LIN {X 0,Y 373.483,Z 447.363,A -85,B 0,C 180,E1 -12862.635,E2 -12862.635} C_VEL
LIN {X 0,Y 372.77,Z 459.424,A -85,B 0,C 180,E1 -12863.505,E2 -12863.505} C_VEL
LIN {X 0,Y 371.923,Z 468.35,A -85,B 0,C 180,E1 -12864.307,E2 -12864.307} C_VEL
LIN {X 0,Y 371.061,Z 479.116,A -85,B 0,C 180,E1 -12865.519,E2 -12865.519} C_VEL
LIN {X 0,Y 370.222,Z 487.926,A -85,B 0,C 180,E1 -12866.736,E2 -12866.736} C_VEL
LIN {X 0,Y 369.443,Z 497.479,A -85,B 0,C 180,E1 -12868.365,E2 -12868.365} C_VEL
LIN {X 0,Y 368.694,Z 505.108,A -85,B 0,C 180,E1 -12870,E2 -12870} C_VEL
LIN {X 0,Y 368.224,Z 511.231,A -85,B 0,C 180,E1 -12871.641,E2 -12871.641} C_VEL
LIN {X 0,Y 367.89,Z 516.098,A -85,B 0,C 180,E1 -12873.286,E2 -12873.286} C_VEL
LIN {X 0,Y 367.719,Z 519.853,A -85,B 0,C 180,E1 -12874.934,E2 -12874.934} C_VEL
LIN {X 0,Y 367.623,Z 522.596,A -85,B 0,C 180,E1 -12876.587,E2 -12876.587} C_VEL
LIN {X 0,Y 367.369,Z 524.811,A -85,B 0,C 180,E1 -12878.804,E2 -12878.804} C_VEL
LIN {X 0,Y 367.305,Z 525.292,A -85,B 0,C 180,E1 -12879.916,E2 -12879.916} C_VEL
LIN {X 0,Y 367.371,Z 525.357,A -85,B 0,C 180,E1 -12881.029,E2 -12881.029} C_VEL
LIN {X 0,Y 367.515,Z 524.674,A -85,B 0,C 180,E1 -12882.768,E2 -12882.768} C_VEL
LIN {X 0,Y 367.623,Z 523.153,A -85,B 0,C 180,E1 -12884.391,E2 -12884.391} C_VEL
LIN {X 0,Y 367.976,Z 520.609,A -85,B 0,C 180,E1 -12886.078,E2 -12886.078} C_VEL
LIN {X 0,Y 368.384,Z 517.012,A -85,B 0,C 180,E1 -12887.773,E2 -12887.773} C_VEL
LIN {X 0,Y 368.981,Z 512.245,A -85,B 0,C 180,E1 -12889.471,E2 -12889.471} C_VEL
LIN {X 0,Y 369.433,Z 508.887,A -85,B 0,C 180,E1 -12890.455,E2 -12890.455} C_VEL
LIN {X 0,Y 369.179,Z 505.977,A -85,B 0,C 180,E1 -12891.251,E2 -12891.251} C_VEL
LIN {X 0,Y 367.085,Z 500.999,A -85,B 0,C 180,E1 -12892.546,E2 -12892.546} C_VEL
LIN {X 0,Y 365.06,Z 495.431,A -85,B 0,C 180,E1 -12893.789,E2 -12893.789} C_VEL
LIN {X 0,Y 364.906,Z 491.596,A -85,B 0,C 180,E1 -12894.493,E2 -12894.493} C_VEL
LIN {X 0,Y 366.14,Z 482.192,A -85,B 0,C 180,E1 -12895.916,E2 -12895.916} C_VEL
LIN {X 0,Y 367.366,Z 471.755,A -85,B 0,C 180,E1 -12897.178,E2 -12897.178} C_VEL
LIN {X 0,Y 368.601,Z 459.913,A -85,B 0,C 180,E1 -12898.313,E2 -12898.313} C_VEL
LIN {X 0,Y 369.641,Z 447.439,A -85,B 0,C 180,E1 -12899.223,E2 -12899.223} C_VEL
LIN {X 0,Y 370.361,Z 434.476,A -85,B 0,C 180,E1 -12899.915,E2 -12899.915} C_VEL
LIN {X 0,Y 370.809,Z 422.498,A -85,B 0,C 180,E1 -12900.346,E2 -12900.346} C_VEL
LIN {X 0,Y 372.684,Z 341.338,A -85,B 0,C 180,E1 -12901.941,E2 -12901.941} C_VEL
LIN {X 0,Y 369.707,Z 328.526,A -85,B 0,C 180,E1 -12902.432,E2 -12902.432} C_VEL
LIN {X 0,Y 364.874,Z 317.06,A -85,B 0,C 180,E1 -12903.049,E2 -12903.049} C_VEL
LIN {X 0,Y 364.019,Z 314.785,A -85,B 0,C 180,E1 -12903.186,E2 -12903.186} C_VEL
LIN {X 0,Y 361.887,Z 305.411,A -85,B 0,C 180,E1 -12905.892,E2 -12905.892} C_VEL
LIN {X 0,Y 361.869,Z 305.412,A -85,B 0,C 180,E1 -12909.027,E2 -12909.027} C_VEL
LIN {X 0,Y 361.835,Z 305.415,A -85,B 0,C 180,E1 -12912.829,E2 -12912.829} C_VEL
LIN {X 0,Y 361.818,Z 305.415,A -85,B 0,C 180,E1 -12915.947,E2 -12915.947} C_VEL
LIN {X 0,Y 361.835,Z 305.412,A -85,B 0,C 180,E1 -12919.245,E2 -12919.245} C_VEL
LIN {X 0,Y 361.863,Z 305.409,A -85,B 0,C 180,E1 -12922.777,E2 -12922.777} C_VEL
LIN {X 0,Y 361.853,Z 305.404,A -85,B 0,C 180,E1 -12925.72,E2 -12925.72} C_VEL
LIN {X 0,Y 361.874,Z 305.401,A -85,B 0,C 180,E1 -12929.672,E2 -12929.672} C_VEL
LIN {X 0,Y 361.953,Z 305.392,A -85,B 0,C 180,E1 -12933.475,E2 -12933.475} C_VEL
LIN {X 0,Y 361.882,Z 305.399,A -85,B 0,C 180,E1 -12937.144,E2 -12937.144} C_VEL
LIN {X 0,Y 361.911,Z 305.393,A -85,B 0,C 180,E1 -12940.724,E2 -12940.724} C_VEL
LIN {X 0,Y 361.933,Z 305.4,A -85,B 0,C 180,E1 -12943.066,E2 -12943.066} C_VEL
LIN {X 0,Y 361.998,Z 305.39,A -85,B 0,C 180,E1 -12946.528,E2 -12946.528} C_VEL
LIN {X 0,Y 362.031,Z 305.387,A -85,B 0,C 180,E1 -12949.938,E2 -12949.938} C_VEL
LIN {X 0,Y 362.15,Z 305.37,A -85,B 0,C 180,E1 -12952.193,E2 -12952.193} C_VEL
LIN {X 0,Y 362.116,Z 305.375,A -85,B 0,C 180,E1 -12954.431,E2 -12954.431} C_VEL
LIN {X 0,Y 362.28,Z 305.352,A -85,B 0,C 180,E1 -12957.777,E2 -12957.777} C_VEL
LIN {X 0,Y 362.426,Z 305.34,A -85,B 0,C 180,E1 -12960,E2 -12960} C_VEL
LIN {X 0,Y 362.28,Z 305.35,A -85,B 0,C 180,E1 -12962.224,E2 -12962.224} C_VEL
LIN {X 0,Y 362.17,Z 305.361,A -85,B 0,C 180,E1 -12966.686,E2 -12966.686} C_VEL
LIN {X 0,Y 362.074,Z 305.38,A -85,B 0,C 180,E1 -12968.933,E2 -12968.933} C_VEL
LIN {X 0,Y 361.96,Z 305.39,A -85,B 0,C 180,E1 -12972.333,E2 -12972.333} C_VEL
LIN {X 0,Y 361.962,Z 305.394,A -85,B 0,C 180,E1 -12974.621,E2 -12974.621} C_VEL
LIN {X 0,Y 361.96,Z 305.395,A -85,B 0,C 180,E1 -12978.1,E2 -12978.1} C_VEL
LIN {X 0,Y 361.862,Z 305.405,A -85,B 0,C 180,E1 -12981.655,E2 -12981.655} C_VEL
LIN {X 0,Y 361.928,Z 305.399,A -85,B 0,C 180,E1 -12985.29,E2 -12985.29} C_VEL
LIN {X 0,Y 361.915,Z 305.398,A -85,B 0,C 180,E1 -12987.779,E2 -12987.779} C_VEL
LIN {X 0,Y 361.847,Z 305.409,A -85,B 0,C 180,E1 -12991.285,E2 -12991.285} C_VEL
LIN {X 0,Y 361.855,Z 305.408,A -85,B 0,C 180,E1 -12994.281,E2 -12994.281} C_VEL
LIN {X 0,Y 361.864,Z 305.41,A -85,B 0,C 180,E1 -12997.223,E2 -12997.223} C_VEL
LIN {X 0,Y 361.836,Z 305.393,A -85,B 0,C 180,E1 -13000.755,E2 -13000.755} C_VEL
LIN {X 0,Y 361.818,Z 305.41,A -85,B 0,C 180,E1 -13004.369,E2 -13004.369} C_VEL
LIN {X 0,Y 361.838,Z 305.415,A -85,B 0,C 180,E1 -13007.568,E2 -13007.568} C_VEL
LIN {X 0,Y 361.87,Z 305.407,A -85,B 0,C 180,E1 -13010.974,E2 -13010.974} C_VEL
LIN {X 0,Y 361.876,Z 305.408,A -85,B 0,C 180,E1 -13014.655,E2 -13014.655} C_VEL
LIN {X 0,Y 361.84,Z 305.414,A -85,B 0,C 180,E1 -13018.371,E2 -13018.371} C_VEL
LIN {X 0,Y 361.876,Z 305.581,A -85,B 0,C 180,E1 -13018.596,E2 -13018.596} C_VEL
LIN {X 0,Y 364.465,Z 316.266,A -85,B 0,C 180,E1 -13021.494,E2 -13021.494} C_VEL
LIN {X 0,Y 366.316,Z 325.27,A -85,B 0,C 180,E1 -13023.815,E2 -13023.815} C_VEL
LIN {X 0,Y 366.607,Z 328.794,A -85,B 0,C 180,E1 -13024.67,E2 -13024.67} C_VEL
LIN {X 0,Y 365.489,Z 339.127,A -85,B 0,C 180,E1 -13027.004,E2 -13027.004} C_VEL
LIN {X 0,Y 370.301,Z 363.459,A -85,B 0,C 180,E1 -13027.884,E2 -13027.884} C_VEL
LIN {X 0,Y 372.048,Z 374.943,A -85,B 0,C 180,E1 -13028.251,E2 -13028.251} C_VEL
LIN {X 0,Y 370.652,Z 448.342,A -85,B 0,C 180,E1 -13029.718,E2 -13029.718} C_VEL
LIN {X 0,Y 369.806,Z 462.108,A -85,B 0,C 180,E1 -13030.213,E2 -13030.213} C_VEL
LIN {X 0,Y 368.828,Z 474.473,A -85,B 0,C 180,E1 -13030.882,E2 -13030.882} C_VEL
LIN {X 0,Y 367.642,Z 486.322,A -85,B 0,C 180,E1 -13031.758,E2 -13031.758} C_VEL
LIN {X 0,Y 366.31,Z 497.713,A -85,B 0,C 180,E1 -13032.843,E2 -13032.843} C_VEL
LIN {X 0,Y 365.033,Z 508.003,A -85,B 0,C 180,E1 -13034.076,E2 -13034.076} C_VEL
LIN {X 0,Y 363.946,Z 517.267,A -85,B 0,C 180,E1 -13035.461,E2 -13035.461} C_VEL
LIN {X 0,Y 362.775,Z 526.272,A -85,B 0,C 180,E1 -13037.127,E2 -13037.127} C_VEL
LIN {X 0,Y 361.748,Z 533.548,A -85,B 0,C 180,E1 -13038.797,E2 -13038.797} C_VEL
LIN {X 0,Y 361.097,Z 539.398,A -85,B 0,C 180,E1 -13040.477,E2 -13040.477} C_VEL
LIN {X 0,Y 360.68,Z 544.022,A -85,B 0,C 180,E1 -13042.16,E2 -13042.16} C_VEL
LIN {X 0,Y 360.433,Z 547.766,A -85,B 0,C 180,E1 -13043.956,E2 -13043.956} C_VEL
LIN {X 0,Y 360.366,Z 550.098,A -85,B 0,C 180,E1 -13045.525,E2 -13045.525} C_VEL
LIN {X 0,Y 360.302,Z 551.291,A -85,B 0,C 180,E1 -13046.645,E2 -13046.645} C_VEL
LIN {X 0,Y 360.359,Z 552.416,A -85,B 0,C 180,E1 -13048.882,E2 -13048.882} C_VEL
LIN {X 0,Y 360.423,Z 552.399,A -85,B 0,C 180,E1 -13050,E2 -13050} C_VEL
LIN {X 0,Y 360.39,Z 551.989,A -85,B 0,C 180,E1 -13051.117,E2 -13051.117} C_VEL
LIN {X 0,Y 360.326,Z 551.137,A -85,B 0,C 180,E1 -13052.235,E2 -13052.235} C_VEL
LIN {X 0,Y 360.323,Z 549.88,A -85,B 0,C 180,E1 -13053.354,E2 -13053.354} C_VEL
LIN {X 0,Y 360.38,Z 547.205,A -85,B 0,C 180,E1 -13055.034,E2 -13055.034} C_VEL
LIN {X 0,Y 360.498,Z 543.495,A -85,B 0,C 180,E1 -13056.717,E2 -13056.717} C_VEL
LIN {X 0,Y 360.74,Z 538.65,A -85,B 0,C 180,E1 -13058.401,E2 -13058.401} C_VEL
LIN {X 0,Y 361.156,Z 532.524,A -85,B 0,C 180,E1 -13060.086,E2 -13060.086} C_VEL
LIN {X 0,Y 361.781,Z 524.896,A -85,B 0,C 180,E1 -13061.769,E2 -13061.769} C_VEL
LIN {X 0,Y 362.498,Z 517.094,A -85,B 0,C 180,E1 -13063.167,E2 -13063.167} C_VEL
LIN {X 0,Y 363.408,Z 507.556,A -85,B 0,C 180,E1 -13064.56,E2 -13064.56} C_VEL
LIN {X 0,Y 364.157,Z 496.934,A -85,B 0,C 180,E1 -13065.819,E2 -13065.819} C_VEL
LIN {X 0,Y 365.223,Z 485.127,A -85,B 0,C 180,E1 -13066.92,E2 -13066.92} C_VEL
LIN {X 0,Y 366.096,Z 473.602,A -85,B 0,C 180,E1 -13067.743,E2 -13067.743} C_VEL
LIN {X 0,Y 366.89,Z 460.601,A -85,B 0,C 180,E1 -13068.425,E2 -13068.425} C_VEL
LIN {X 0,Y 367.493,Z 448.03,A -85,B 0,C 180,E1 -13068.863,E2 -13068.863} C_VEL
LIN {X 0,Y 368.551,Z 374.347,A -85,B 0,C 180,E1 -13070.314,E2 -13070.314} C_VEL
LIN {X 0,Y 363.817,Z 339.576,A -85,B 0,C 180,E1 -13071.265,E2 -13071.265} C_VEL
LIN {X 0,Y 365.161,Z 323.765,A -85,B 0,C 180,E1 -13074.746,E2 -13074.746} C_VEL
LIN {X 0,Y 364.791,Z 319.684,A -85,B 0,C 180,E1 -13075.692,E2 -13075.692} C_VEL
LIN {X 0,Y 362.335,Z 307.335,A -85,B 0,C 180,E1 -13078.689,E2 -13078.689} C_VEL
LIN {X 0,Y 361.935,Z 305.401,A -85,B 0,C 180,E1 -13079.184,E2 -13079.184} C_VEL
LIN {X 0,Y 361.858,Z 305.406,A -85,B 0,C 180,E1 -13083.369,E2 -13083.369} C_VEL
LIN {X 0,Y 361.866,Z 305.406,A -85,B 0,C 180,E1 -13087.017,E2 -13087.017} C_VEL
LIN {X 0,Y 361.853,Z 305.409,A -85,B 0,C 180,E1 -13089.861,E2 -13089.861} C_VEL
LIN {X 0,Y 361.834,Z 305.412,A -85,B 0,C 180,E1 -13092.828,E2 -13092.828} C_VEL
LIN {X 0,Y 361.816,Z 305.413,A -85,B 0,C 180,E1 -13095.946,E2 -13095.946} C_VEL
LIN {X 0,Y 361.833,Z 305.41,A -85,B 0,C 180,E1 -13099.244,E2 -13099.244} C_VEL
LIN {X 0,Y 361.861,Z 305.412,A -85,B 0,C 180,E1 -13102.776,E2 -13102.776} C_VEL
LIN {X 0,Y 361.851,Z 305.407,A -85,B 0,C 180,E1 -13105.719,E2 -13105.719} C_VEL
LIN {X 0,Y 361.869,Z 305.405,A -85,B 0,C 180,E1 -13109.671,E2 -13109.671} C_VEL
LIN {X 0,Y 361.95,Z 305.397,A -85,B 0,C 180,E1 -13113.474,E2 -13113.474} C_VEL
LIN {X 0,Y 361.886,Z 305.409,A -85,B 0,C 180,E1 -13117.144,E2 -13117.144} C_VEL
LIN {X 0,Y 361.917,Z 305.401,A -85,B 0,C 180,E1 -13120.724,E2 -13120.724} C_VEL
LIN {X 0,Y 361.942,Z 305.396,A -85,B 0,C 180,E1 -13124.226,E2 -13124.226} C_VEL
LIN {X 0,Y 361.994,Z 305.389,A -85,B 0,C 180,E1 -13126.527,E2 -13126.527} C_VEL
LIN {X 0,Y 362.027,Z 305.387,A -85,B 0,C 180,E1 -13129.938,E2 -13129.938} C_VEL
LIN {X 0,Y 362.157,Z 305.373,A -85,B 0,C 180,E1 -13133.313,E2 -13133.313} C_VEL
LIN {X 0,Y 362.275,Z 305.36,A -85,B 0,C 180,E1 -13137.776,E2 -13137.776} C_VEL
LIN {X 0,Y 362.421,Z 305.34,A -85,B 0,C 180,E1 -13140,E2 -13140} C_VEL
LIN {X 0,Y 362.276,Z 305.356,A -85,B 0,C 180,E1 -13142.223,E2 -13142.223} C_VEL
LIN {X 0,Y 362.134,Z 305.372,A -85,B 0,C 180,E1 -13146.687,E2 -13146.687} C_VEL
LIN {X 0,Y 362.026,Z 305.392,A -85,B 0,C 180,E1 -13150.062,E2 -13150.062} C_VEL
LIN {X 0,Y 361.993,Z 305.394,A -85,B 0,C 180,E1 -13153.899,E2 -13153.899} C_VEL
LIN {X 0,Y 361.962,Z 305.397,A -85,B 0,C 180,E1 -13157.939,E2 -13157.939} C_VEL
LIN {X 0,Y 361.856,Z 305.407,A -85,B 0,C 180,E1 -13161.655,E2 -13161.655} C_VEL
LIN {X 0,Y 361.921,Z 305.399,A -85,B 0,C 180,E1 -13165.29,E2 -13165.29} C_VEL
LIN {X 0,Y 361.913,Z 305.4,A -85,B 0,C 180,E1 -13167.778,E2 -13167.778} C_VEL
LIN {X 0,Y 361.842,Z 305.409,A -85,B 0,C 180,E1 -13171.285,E2 -13171.285} C_VEL
LIN {X 0,Y 361.849,Z 305.41,A -85,B 0,C 180,E1 -13174.281,E2 -13174.281} C_VEL
LIN {X 0,Y 361.858,Z 305.408,A -85,B 0,C 180,E1 -13177.223,E2 -13177.223} C_VEL
LIN {X 0,Y 361.831,Z 305.416,A -85,B 0,C 180,E1 -13180.756,E2 -13180.756} C_VEL
LIN {X 0,Y 361.812,Z 305.413,A -85,B 0,C 180,E1 -13184.369,E2 -13184.369} C_VEL
LIN {X 0,Y 361.825,Z 305.412,A -85,B 0,C 180,E1 -13187.57,E2 -13187.57} C_VEL
LIN {X 0,Y 361.84,Z 305.411,A -85,B 0,C 180,E1 -13191.573,E2 -13191.573} C_VEL
LIN {X 0,Y 361.871,Z 305.406,A -85,B 0,C 180,E1 -13194.656,E2 -13194.656} C_VEL
LIN {X 0,Y 361.834,Z 305.409,A -85,B 0,C 180,E1 -13198.371,E2 -13198.371} C_VEL
LIN {X 0,Y 361.863,Z 305.408,A -85,B 0,C 180,E1 -13200.953,E2 -13200.953} C_VEL
LIN {X 0,Y 361.863,Z 305.406,A -85,B 0,C 180,E1 -13204.706,E2 -13204.706} C_VEL
LIN {X 0,Y 361.859,Z 305.407,A -85,B 0,C 180,E1 -13208.346,E2 -13208.346} C_VEL
LIN {X 0,Y 361.919,Z 305.401,A -85,B 0,C 180,E1 -13212.085,E2 -13212.085} C_VEL
LIN {X 0,Y 361.961,Z 305.397,A -85,B 0,C 180,E1 -13215.38,E2 -13215.38} C_VEL
LIN {X 0,Y 362.044,Z 305.52,A -85,B 0,C 180,E1 -13216.471,E2 -13216.471} C_VEL
LIN {X 0,Y 363.735,Z 314.698,A -85,B 0,C 180,E1 -13218.825,E2 -13218.825} C_VEL
LIN {X 0,Y 366.129,Z 323.28,A -85,B 0,C 180,E1 -13219.123,E2 -13219.123} C_VEL
LIN {X 0,Y 369.003,Z 340.775,A -85,B 0,C 180,E1 -13219.62,E2 -13219.62} C_VEL
LIN {X 0,Y 367.65,Z 421.709,A -85,B 0,C 180,E1 -13221.204,E2 -13221.204} C_VEL
LIN {X 0,Y 367.211,Z 434.918,A -85,B 0,C 180,E1 -13221.678,E2 -13221.678} C_VEL
LIN {X 0,Y 366.63,Z 447.574,A -85,B 0,C 180,E1 -13222.358,E2 -13222.358} C_VEL
LIN {X 0,Y 365.897,Z 459.648,A -85,B 0,C 180,E1 -13223.244,E2 -13223.244} C_VEL
LIN {X 0,Y 365.012,Z 468.583,A -85,B 0,C 180,E1 -13224.06,E2 -13224.06} C_VEL
LIN {X 0,Y 364.125,Z 479.354,A -85,B 0,C 180,E1 -13225.295,E2 -13225.295} C_VEL
LIN {X 0,Y 363.193,Z 489.05,A -85,B 0,C 180,E1 -13226.672,E2 -13226.672} C_VEL
LIN {X 0,Y 362.499,Z 496.99,A -85,B 0,C 180,E1 -13228.056,E2 -13228.056} C_VEL
LIN {X 0,Y 361.721,Z 504.802,A -85,B 0,C 180,E1 -13229.722,E2 -13229.722} C_VEL
LIN {X 0,Y 361.258,Z 510.097,A -85,B 0,C 180,E1 -13231.115,E2 -13231.115} C_VEL
LIN {X 0,Y 360.914,Z 515.27,A -85,B 0,C 180,E1 -13232.791,E2 -13232.791} C_VEL
LIN {X 0,Y 360.627,Z 519.299,A -85,B 0,C 180,E1 -13234.471,E2 -13234.471} C_VEL
LIN {X 0,Y 360.589,Z 522.465,A -85,B 0,C 180,E1 -13236.278,E2 -13236.278} C_VEL
LIN {X 0,Y 360.357,Z 524.306,A -85,B 0,C 180,E1 -13237.847,E2 -13237.847} C_VEL
LIN {X 0,Y 360.255,Z 525.162,A -85,B 0,C 180,E1 -13238.979,E2 -13238.979} C_VEL
LIN {X 0,Y 360.314,Z 525.604,A -85,B 0,C 180,E1 -13241.248,E2 -13241.248} C_VEL
LIN {X 0,Y 360.443,Z 524.953,A -85,B 0,C 180,E1 -13242.862,E2 -13242.862} C_VEL
LIN {X 0,Y 360.598,Z 523.239,A -85,B 0,C 180,E1 -13244.677,E2 -13244.677} C_VEL
LIN {X 0,Y 360.959,Z 520.611,A -85,B 0,C 180,E1 -13246.399,E2 -13246.399} C_VEL
LIN {X 0,Y 361.435,Z 516.923,A -85,B 0,C 180,E1 -13248.127,E2 -13248.127} C_VEL
LIN {X 0,Y 362.065,Z 512.058,A -85,B 0,C 180,E1 -13249.858,E2 -13249.858} C_VEL
LIN {X 0,Y 362.941,Z 505.631,A -85,B 0,C 180,E1 -13251.648,E2 -13251.648} C_VEL
LIN {X 0,Y 363.969,Z 498.087,A -85,B 0,C 180,E1 -13253.319,E2 -13253.319} C_VEL
LIN {X 0,Y 364.906,Z 491.596,A -85,B 0,C 180,E1 -13254.493,E2 -13254.493} C_VEL
LIN {X 0,Y 364.796,Z 487.582,A -85,B 0,C 180,E1 -13255.176,E2 -13255.176} C_VEL
LIN {X 0,Y 362.993,Z 480.92,A -85,B 0,C 180,E1 -13256.299,E2 -13256.299} C_VEL
LIN {X 0,Y 361.199,Z 473.773,A -85,B 0,C 180,E1 -13257.344,E2 -13257.344} C_VEL
LIN {X 0,Y 361.086,Z 469.006,A -85,B 0,C 180,E1 -13257.894,E2 -13257.894} C_VEL
LIN {X 0,Y 362.176,Z 458.535,A -85,B 0,C 180,E1 -13258.862,E2 -13258.862} C_VEL
LIN {X 0,Y 363.184,Z 446.482,A -85,B 0,C 180,E1 -13259.726,E2 -13259.726} C_VEL
LIN {X 0,Y 363.944,Z 433.308,A -85,B 0,C 180,E1 -13260.418,E2 -13260.418} C_VEL
LIN {X 0,Y 364.313,Z 422.973,A -85,B 0,C 180,E1 -13260.785,E2 -13260.785} C_VEL
LIN {X 0,Y 366.246,Z 342.244,A -85,B 0,C 180,E1 -13262.4,E2 -13262.4} C_VEL
LIN {X 0,Y 363.71,Z 331.264,A -85,B 0,C 180,E1 -13262.832,E2 -13262.832} C_VEL
LIN {X 0,Y 356.879,Z 315.033,A -85,B 0,C 180,E1 -13263.772,E2 -13263.772} C_VEL
LIN {X 0,Y 354.848,Z 306.282,A -85,B 0,C 180,E1 -13266.35,E2 -13266.35} C_VEL
LIN {X 0,Y 354.824,Z 306.288,A -85,B 0,C 180,E1 -13269.424,E2 -13269.424} C_VEL
LIN {X 0,Y 354.787,Z 306.293,A -85,B 0,C 180,E1 -13272.867,E2 -13272.867} C_VEL
LIN {X 0,Y 354.766,Z 306.294,A -85,B 0,C 180,E1 -13276.104,E2 -13276.104} C_VEL
LIN {X 0,Y 354.788,Z 306.29,A -85,B 0,C 180,E1 -13279.179,E2 -13279.179} C_VEL
LIN {X 0,Y 354.807,Z 306.285,A -85,B 0,C 180,E1 -13282.403,E2 -13282.403} C_VEL
LIN {X 0,Y 354.811,Z 306.285,A -85,B 0,C 180,E1 -13284.941,E2 -13284.941} C_VEL
LIN {X 0,Y 354.793,Z 306.283,A -85,B 0,C 180,E1 -13288.405,E2 -13288.405} C_VEL
LIN {X 0,Y 354.848,Z 306.274,A -85,B 0,C 180,E1 -13291.619,E2 -13291.619} C_VEL
LIN {X 0,Y 354.898,Z 306.27,A -85,B 0,C 180,E1 -13294.173,E2 -13294.173} C_VEL
LIN {X 0,Y 354.816,Z 306.284,A -85,B 0,C 180,E1 -13297.893,E2 -13297.893} C_VEL
LIN {X 0,Y 354.922,Z 306.274,A -85,B 0,C 180,E1 -13301.892,E2 -13301.892} C_VEL
LIN {X 0,Y 354.943,Z 306.272,A -85,B 0,C 180,E1 -13305.981,E2 -13305.981} C_VEL
LIN {X 0,Y 354.977,Z 306.263,A -85,B 0,C 180,E1 -13309.736,E2 -13309.736} C_VEL
LIN {X 0,Y 355.113,Z 306.248,A -85,B 0,C 180,E1 -13312.037,E2 -13312.037} C_VEL
LIN {X 0,Y 355.091,Z 306.251,A -85,B 0,C 180,E1 -13314.321,E2 -13314.321} C_VEL
LIN {X 0,Y 355.244,Z 306.228,A -85,B 0,C 180,E1 -13317.733,E2 -13317.733} C_VEL
LIN {X 0,Y 355.375,Z 306.218,A -85,B 0,C 180,E1 -13320,E2 -13320} C_VEL
LIN {X 0,Y 355.243,Z 306.226,A -85,B 0,C 180,E1 -13322.268,E2 -13322.268} C_VEL
LIN {X 0,Y 355.137,Z 306.236,A -85,B 0,C 180,E1 -13326.819,E2 -13326.819} C_VEL
LIN {X 0,Y 355.015,Z 306.258,A -85,B 0,C 180,E1 -13329.113,E2 -13329.113} C_VEL
LIN {X 0,Y 354.921,Z 306.269,A -85,B 0,C 180,E1 -13332.581,E2 -13332.581} C_VEL
LIN {X 0,Y 354.89,Z 306.27,A -85,B 0,C 180,E1 -13336.096,E2 -13336.096} C_VEL
LIN {X 0,Y 354.907,Z 306.277,A -85,B 0,C 180,E1 -13338.472,E2 -13338.472} C_VEL
LIN {X 0,Y 354.818,Z 306.284,A -85,B 0,C 180,E1 -13342.107,E2 -13342.107} C_VEL
LIN {X 0,Y 354.899,Z 306.273,A -85,B 0,C 180,E1 -13345.828,E2 -13345.828} C_VEL
LIN {X 0,Y 354.855,Z 306.28,A -85,B 0,C 180,E1 -13349.679,E2 -13349.679} C_VEL
LIN {X 0,Y 354.807,Z 306.287,A -85,B 0,C 180,E1 -13353.702,E2 -13353.702} C_VEL
LIN {X 0,Y 354.798,Z 306.283,A -85,B 0,C 180,E1 -13356.46,E2 -13356.46} C_VEL
LIN {X 0,Y 354.825,Z 306.271,A -85,B 0,C 180,E1 -13359.424,E2 -13359.424} C_VEL
LIN {X 0,Y 354.79,Z 306.289,A -85,B 0,C 180,E1 -13362.867,E2 -13362.867} C_VEL
LIN {X 0,Y 354.768,Z 306.292,A -85,B 0,C 180,E1 -13366.104,E2 -13366.104} C_VEL
LIN {X 0,Y 354.789,Z 306.29,A -85,B 0,C 180,E1 -13369.179,E2 -13369.179} C_VEL
LIN {X 0,Y 354.809,Z 306.282,A -85,B 0,C 180,E1 -13372.403,E2 -13372.403} C_VEL
LIN {X 0,Y 354.814,Z 306.286,A -85,B 0,C 180,E1 -13374.941,E2 -13374.941} C_VEL
LIN {X 0,Y 354.794,Z 306.387,A -85,B 0,C 180,E1 -13378.087,E2 -13378.087} C_VEL
LIN {X 0,Y 357.582,Z 317.605,A -85,B 0,C 180,E1 -13381.215,E2 -13381.215} C_VEL
LIN {X 0,Y 359.685,Z 328.237,A -85,B 0,C 180,E1 -13384.003,E2 -13384.003} C_VEL
LIN {X 0,Y 359.409,Z 333.05,A -85,B 0,C 180,E1 -13385.139,E2 -13385.139} C_VEL
LIN {X 0,Y 358.771,Z 338.826,A -85,B 0,C 180,E1 -13386.469,E2 -13386.469} C_VEL
LIN {X 0,Y 363.58,Z 362.705,A -85,B 0,C 180,E1 -13387.371,E2 -13387.371} C_VEL
LIN {X 0,Y 365.621,Z 376.5,A -85,B 0,C 180,E1 -13387.819,E2 -13387.819} C_VEL
LIN {X 0,Y 364.145,Z 447.901,A -85,B 0,C 180,E1 -13389.265,E2 -13389.265} C_VEL
LIN {X 0,Y 363.291,Z 461.72,A -85,B 0,C 180,E1 -13389.769,E2 -13389.769} C_VEL
LIN {X 0,Y 362.275,Z 474.114,A -85,B 0,C 180,E1 -13390.449,E2 -13390.449} C_VEL
LIN {X 0,Y 361.141,Z 485.193,A -85,B 0,C 180,E1 -13391.27,E2 -13391.27} C_VEL
LIN {X 0,Y 359.721,Z 496.737,A -85,B 0,C 180,E1 -13392.372,E2 -13392.372} C_VEL
LIN {X 0,Y 358.346,Z 507.144,A -85,B 0,C 180,E1 -13393.624,E2 -13393.624} C_VEL
LIN {X 0,Y 357.23,Z 515.967,A -85,B 0,C 180,E1 -13394.939,E2 -13394.939} C_VEL
LIN {X 0,Y 356.011,Z 524.944,A -85,B 0,C 180,E1 -13396.587,E2 -13396.587} C_VEL
LIN {X 0,Y 354.909,Z 532.405,A -85,B 0,C 180,E1 -13398.289,E2 -13398.289} C_VEL
LIN {X 0,Y 354.061,Z 539.321,A -85,B 0,C 180,E1 -13400.286,E2 -13400.286} C_VEL
LIN {X 0,Y 353.624,Z 543.903,A -85,B 0,C 180,E1 -13402.003,E2 -13402.003} C_VEL
LIN {X 0,Y 353.325,Z 547.893,A -85,B 0,C 180,E1 -13404.019,E2 -13404.019} C_VEL
LIN {X 0,Y 353.279,Z 549.911,A -85,B 0,C 180,E1 -13405.436,E2 -13405.436} C_VEL
LIN {X 0,Y 353.223,Z 551.073,A -85,B 0,C 180,E1 -13406.578,E2 -13406.578} C_VEL
LIN {X 0,Y 353.26,Z 552.159,A -85,B 0,C 180,E1 -13408.86,E2 -13408.86} C_VEL
LIN {X 0,Y 353.328,Z 552.126,A -85,B 0,C 180,E1 -13410,E2 -13410} C_VEL
LIN {X 0,Y 353.292,Z 551.688,A -85,B 0,C 180,E1 -13411.139,E2 -13411.139} C_VEL
LIN {X 0,Y 353.245,Z 549.537,A -85,B 0,C 180,E1 -13413.421,E2 -13413.421} C_VEL
LIN {X 0,Y 353.283,Z 546.823,A -85,B 0,C 180,E1 -13415.136,E2 -13415.136} C_VEL
LIN {X 0,Y 353.416,Z 543.073,A -85,B 0,C 180,E1 -13416.852,E2 -13416.852} C_VEL
LIN {X 0,Y 353.679,Z 538.186,A -85,B 0,C 180,E1 -13418.57,E2 -13418.57} C_VEL
LIN {X 0,Y 354.121,Z 532.014,A -85,B 0,C 180,E1 -13420.289,E2 -13420.289} C_VEL
LIN {X 0,Y 354.802,Z 524.33,A -85,B 0,C 180,E1 -13422.004,E2 -13422.004} C_VEL
LIN {X 0,Y 355.518,Z 516.45,A -85,B 0,C 180,E1 -13423.431,E2 -13423.431} C_VEL
LIN {X 0,Y 356.439,Z 506.815,A -85,B 0,C 180,E1 -13424.852,E2 -13424.852} C_VEL
LIN {X 0,Y 357.342,Z 496.108,A -85,B 0,C 180,E1 -13426.129,E2 -13426.129} C_VEL
LIN {X 0,Y 358.248,Z 485.776,A -85,B 0,C 180,E1 -13427.113,E2 -13427.113} C_VEL
LIN {X 0,Y 359.218,Z 473.482,A -85,B 0,C 180,E1 -13428.021,E2 -13428.021} C_VEL
LIN {X 0,Y 360.054,Z 460.535,A -85,B 0,C 180,E1 -13428.714,E2 -13428.714} C_VEL
LIN {X 0,Y 360.663,Z 448.059,A -85,B 0,C 180,E1 -13429.16,E2 -13429.16} C_VEL
LIN {X 0,Y 361.71,Z 373.95,A -85,B 0,C 180,E1 -13430.653,E2 -13430.653} C_VEL
LIN {X 0,Y 356.886,Z 339.268,A -85,B 0,C 180,E1 -13431.638,E2 -13431.638} C_VEL
LIN {X 0,Y 358.206,Z 324.519,A -85,B 0,C 180,E1 -13434.949,E2 -13434.949} C_VEL
LIN {X 0,Y 357.487,Z 319.076,A -85,B 0,C 180,E1 -13436.252,E2 -13436.252} C_VEL
LIN {X 0,Y 354.917,Z 306.486,A -85,B 0,C 180,E1 -13439.392,E2 -13439.392} C_VEL
LIN {X 0,Y 354.87,Z 306.281,A -85,B 0,C 180,E1 -13439.676,E2 -13439.676} C_VEL
LIN {X 0,Y 354.806,Z 306.287,A -85,B 0,C 180,E1 -13443.701,E2 -13443.701} C_VEL
LIN {X 0,Y 354.797,Z 306.29,A -85,B 0,C 180,E1 -13446.459,E2 -13446.459} C_VEL
LIN {X 0,Y 354.823,Z 306.283,A -85,B 0,C 180,E1 -13449.423,E2 -13449.423} C_VEL
LIN {X 0,Y 354.786,Z 306.29,A -85,B 0,C 180,E1 -13452.866,E2 -13452.866} C_VEL
LIN {X 0,Y 354.765,Z 306.292,A -85,B 0,C 180,E1 -13456.103,E2 -13456.103} C_VEL
LIN {X 0,Y 354.786,Z 306.289,A -85,B 0,C 180,E1 -13459.178,E2 -13459.178} C_VEL
LIN {X 0,Y 354.805,Z 306.288,A -85,B 0,C 180,E1 -13462.402,E2 -13462.402} C_VEL
LIN {X 0,Y 354.809,Z 306.289,A -85,B 0,C 180,E1 -13464.94,E2 -13464.94} C_VEL
LIN {X 0,Y 354.79,Z 306.289,A -85,B 0,C 180,E1 -13468.404,E2 -13468.404} C_VEL
LIN {X 0,Y 354.843,Z 306.281,A -85,B 0,C 180,E1 -13471.618,E2 -13471.618} C_VEL
LIN {X 0,Y 354.895,Z 306.274,A -85,B 0,C 180,E1 -13474.172,E2 -13474.172} C_VEL
LIN {X 0,Y 354.831,Z 306.282,A -85,B 0,C 180,E1 -13477.893,E2 -13477.893} C_VEL
LIN {X 0,Y 354.919,Z 306.271,A -85,B 0,C 180,E1 -13481.891,E2 -13481.891} C_VEL
LIN {X 0,Y 354.938,Z 306.269,A -85,B 0,C 180,E1 -13485.981,E2 -13485.981} C_VEL
LIN {X 0,Y 354.973,Z 306.267,A -85,B 0,C 180,E1 -13489.736,E2 -13489.736} C_VEL
LIN {X 0,Y 355.122,Z 306.248,A -85,B 0,C 180,E1 -13493.18,E2 -13493.18} C_VEL
LIN {X 0,Y 355.238,Z 306.237,A -85,B 0,C 180,E1 -13497.732,E2 -13497.732} C_VEL
LIN {X 0,Y 355.37,Z 306.218,A -85,B 0,C 180,E1 -13500,E2 -13500} C_VEL
LIN {X 0,Y 355.239,Z 306.233,A -85,B 0,C 180,E1 -13502.267,E2 -13502.267} C_VEL
LIN {X 0,Y 355.098,Z 306.248,A -85,B 0,C 180,E1 -13506.82,E2 -13506.82} C_VEL
LIN {X 0,Y 354.973,Z 306.268,A -85,B 0,C 180,E1 -13510.264,E2 -13510.264} C_VEL
LIN {X 0,Y 354.938,Z 306.274,A -85,B 0,C 180,E1 -13514.019,E2 -13514.019} C_VEL
LIN {X 0,Y 354.917,Z 306.276,A -85,B 0,C 180,E1 -13518.109,E2 -13518.109} C_VEL
LIN {X 0,Y 354.81,Z 306.289,A -85,B 0,C 180,E1 -13522.107,E2 -13522.107} C_VEL
LIN {X 0,Y 354.893,Z 306.275,A -85,B 0,C 180,E1 -13525.828,E2 -13525.828} C_VEL
LIN {X 0,Y 354.849,Z 306.28,A -85,B 0,C 180,E1 -13529.679,E2 -13529.679} C_VEL
LIN {X 0,Y 354.801,Z 306.285,A -85,B 0,C 180,E1 -13533.702,E2 -13533.702} C_VEL
LIN {X 0,Y 354.793,Z 306.29,A -85,B 0,C 180,E1 -13536.46,E2 -13536.46} C_VEL
LIN {X 0,Y 354.82,Z 306.284,A -85,B 0,C 180,E1 -13539.424,E2 -13539.424} C_VEL
LIN {X 0,Y 354.783,Z 306.294,A -85,B 0,C 180,E1 -13542.868,E2 -13542.868} C_VEL
LIN {X 0,Y 354.761,Z 306.29,A -85,B 0,C 180,E1 -13546.104,E2 -13546.104} C_VEL
LIN {X 0,Y 354.762,Z 306.296,A -85,B 0,C 180,E1 -13549.176,E2 -13549.176} C_VEL
LIN {X 0,Y 354.797,Z 306.286,A -85,B 0,C 180,E1 -13552.404,E2 -13552.404} C_VEL
LIN {X 0,Y 354.809,Z 306.288,A -85,B 0,C 180,E1 -13554.941,E2 -13554.941} C_VEL
LIN {X 0,Y 354.79,Z 306.287,A -85,B 0,C 180,E1 -13558.406,E2 -13558.406} C_VEL
LIN {X 0,Y 354.794,Z 306.291,A -85,B 0,C 180,E1 -13561.615,E2 -13561.615} C_VEL
LIN {X 0,Y 354.803,Z 306.291,A -85,B 0,C 180,E1 -13565.42,E2 -13565.42} C_VEL
LIN {X 0,Y 354.825,Z 306.284,A -85,B 0,C 180,E1 -13569.114,E2 -13569.114} C_VEL
LIN {X 0,Y 354.878,Z 306.276,A -85,B 0,C 180,E1 -13572.72,E2 -13572.72} C_VEL
LIN {X 0,Y 354.974,Z 306.412,A -85,B 0,C 180,E1 -13576.216,E2 -13576.216} C_VEL
LIN {X 0,Y 356.56,Z 314.765,A -85,B 0,C 180,E1 -13578.438,E2 -13578.438} C_VEL
LIN {X 0,Y 359.384,Z 324.267,A -85,B 0,C 180,E1 -13578.794,E2 -13578.794} C_VEL
LIN {X 0,Y 362.203,Z 340.303,A -85,B 0,C 180,E1 -13579.27,E2 -13579.27} C_VEL
LIN {X 0,Y 360.834,Z 422.967,A -85,B 0,C 180,E1 -13580.93,E2 -13580.93} C_VEL
LIN {X 0,Y 360.327,Z 436.611,A -85,B 0,C 180,E1 -13581.448,E2 -13581.448} C_VEL
LIN {X 0,Y 359.762,Z 448.868,A -85,B 0,C 180,E1 -13582.141,E2 -13582.141} C_VEL
LIN {X 0,Y 358.92,Z 461.44,A -85,B 0,C 180,E1 -13583.112,E2 -13583.112} C_VEL
LIN {X 0,Y 357.736,Z 472.684,A -85,B 0,C 180,E1 -13584.222,E2 -13584.222} C_VEL
LIN {X 0,Y 356.847,Z 482.758,A -85,B 0,C 180,E1 -13585.482,E2 -13585.482} C_VEL
LIN {X 0,Y 356.01,Z 491.835,A -85,B 0,C 180,E1 -13586.888,E2 -13586.888} C_VEL
LIN {X 0,Y 355.193,Z 500.684,A -85,B 0,C 180,E1 -13588.583,E2 -13588.583} C_VEL
LIN {X 0,Y 354.465,Z 507.825,A -85,B 0,C 180,E1 -13590.284,E2 -13590.284} C_VEL
LIN {X 0,Y 354.066,Z 512.637,A -85,B 0,C 180,E1 -13591.707,E2 -13591.707} C_VEL
LIN {X 0,Y 353.659,Z 517.326,A -85,B 0,C 180,E1 -13593.418,E2 -13593.418} C_VEL
LIN {X 0,Y 353.552,Z 520.902,A -85,B 0,C 180,E1 -13595.132,E2 -13595.132} C_VEL
LIN {X 0,Y 353.385,Z 523.486,A -85,B 0,C 180,E1 -13596.854,E2 -13596.854} C_VEL
LIN {X 0,Y 353.257,Z 524.709,A -85,B 0,C 180,E1 -13598.006,E2 -13598.006} C_VEL
LIN {X 0,Y 353.152,Z 525.489,A -85,B 0,C 180,E1 -13599.161,E2 -13599.161} C_VEL
LIN {X 0,Y 353.228,Z 525.851,A -85,B 0,C 180,E1 -13601.477,E2 -13601.477} C_VEL
LIN {X 0,Y 353.367,Z 525.236,A -85,B 0,C 180,E1 -13602.956,E2 -13602.956} C_VEL
LIN {X 0,Y 353.556,Z 523.327,A -85,B 0,C 180,E1 -13604.976,E2 -13604.976} C_VEL
LIN {X 0,Y 353.965,Z 520.613,A -85,B 0,C 180,E1 -13606.732,E2 -13606.732} C_VEL
LIN {X 0,Y 354.473,Z 516.834,A -85,B 0,C 180,E1 -13608.495,E2 -13608.495} C_VEL
LIN {X 0,Y 355.179,Z 511.872,A -85,B 0,C 180,E1 -13610.26,E2 -13610.26} C_VEL
LIN {X 0,Y 356.102,Z 505.571,A -85,B 0,C 180,E1 -13612.023,E2 -13612.023} C_VEL
LIN {X 0,Y 357.252,Z 497.621,A -85,B 0,C 180,E1 -13613.784,E2 -13613.784} C_VEL
LIN {X 0,Y 358.46,Z 489.433,A -85,B 0,C 180,E1 -13615.242,E2 -13615.242} C_VEL
LIN {X 0,Y 359.815,Z 479.374,A -85,B 0,C 180,E1 -13616.695,E2 -13616.695} C_VEL
LIN {X 0,Y 361.086,Z 469.006,A -85,B 0,C 180,E1 -13617.894,E2 -13617.894} C_VEL
LIN {X 0,Y 361.011,Z 464.093,A -85,B 0,C 180,E1 -13618.418,E2 -13618.418} C_VEL
LIN {X 0,Y 359.181,Z 456.022,A -85,B 0,C 180,E1 -13619.286,E2 -13619.286} C_VEL
LIN {X 0,Y 357.256,Z 447.646,A -85,B 0,C 180,E1 -13620.07,E2 -13620.07} C_VEL
LIN {X 0,Y 356.93,Z 442.233,A -85,B 0,C 180,E1 -13620.442,E2 -13620.442} C_VEL
LIN {X 0,Y 357.585,Z 429.025,A -85,B 0,C 180,E1 -13621.059,E2 -13621.059} C_VEL
LIN {X 0,Y 358.17,Z 416.014,A -85,B 0,C 180,E1 -13621.414,E2 -13621.414} C_VEL
LIN {X 0,Y 359.831,Z 343.242,A -85,B 0,C 180,E1 -13622.876,E2 -13622.876} C_VEL
LIN {X 0,Y 357.527,Z 333.571,A -85,B 0,C 180,E1 -13623.274,E2 -13623.274} C_VEL
LIN {X 0,Y 350.66,Z 317.742,A -85,B 0,C 180,E1 -13624.205,E2 -13624.205} C_VEL
LIN {X 0,Y 349.699,Z 315.318,A -85,B 0,C 180,E1 -13624.379,E2 -13624.379} C_VEL
LIN {X 0,Y 347.758,Z 307.16,A -85,B 0,C 180,E1 -13626.833,E2 -13626.833} C_VEL
LIN {X 0,Y 347.732,Z 307.17,A -85,B 0,C 180,E1 -13630.297,E2 -13630.297} C_VEL
LIN {X 0,Y 347.722,Z 307.171,A -85,B 0,C 180,E1 -13633.408,E2 -13633.408} C_VEL
LIN {X 0,Y 347.725,Z 307.173,A -85,B 0,C 180,E1 -13636.686,E2 -13636.686} C_VEL
LIN {X 0,Y 347.747,Z 307.166,A -85,B 0,C 180,E1 -13640.173,E2 -13640.173} C_VEL
LIN {X 0,Y 347.761,Z 307.165,A -85,B 0,C 180,E1 -13642.679,E2 -13642.679} C_VEL
LIN {X 0,Y 347.748,Z 307.161,A -85,B 0,C 180,E1 -13645.956,E2 -13645.956} C_VEL
LIN {X 0,Y 347.763,Z 307.158,A -85,B 0,C 180,E1 -13649.654,E2 -13649.654} C_VEL
LIN {X 0,Y 347.85,Z 307.144,A -85,B 0,C 180,E1 -13652.745,E2 -13652.745} C_VEL
LIN {X 0,Y 347.785,Z 307.151,A -85,B 0,C 180,E1 -13656.162,E2 -13656.162} C_VEL
LIN {X 0,Y 347.808,Z 307.151,A -85,B 0,C 180,E1 -13659.909,E2 -13659.909} C_VEL
LIN {X 0,Y 347.866,Z 307.151,A -85,B 0,C 180,E1 -13662.359,E2 -13662.359} C_VEL
LIN {X 0,Y 347.897,Z 307.15,A -85,B 0,C 180,E1 -13665.971,E2 -13665.971} C_VEL
LIN {X 0,Y 347.928,Z 307.139,A -85,B 0,C 180,E1 -13669.526,E2 -13669.526} C_VEL
LIN {X 0,Y 348.073,Z 307.127,A -85,B 0,C 180,E1 -13671.875,E2 -13671.875} C_VEL
LIN {X 0,Y 348.066,Z 307.124,A -85,B 0,C 180,E1 -13674.206,E2 -13674.206} C_VEL
LIN {X 0,Y 348.206,Z 307.105,A -85,B 0,C 180,E1 -13677.687,E2 -13677.687} C_VEL
LIN {X 0,Y 348.325,Z 307.096,A -85,B 0,C 180,E1 -13680,E2 -13680} C_VEL
LIN {X 0,Y 348.206,Z 307.102,A -85,B 0,C 180,E1 -13682.314,E2 -13682.314} C_VEL
LIN {X 0,Y 348.105,Z 307.111,A -85,B 0,C 180,E1 -13686.958,E2 -13686.958} C_VEL
LIN {X 0,Y 347.968,Z 307.136,A -85,B 0,C 180,E1 -13689.299,E2 -13689.299} C_VEL
LIN {X 0,Y 347.89,Z 307.148,A -85,B 0,C 180,E1 -13692.84,E2 -13692.84} C_VEL
LIN {X 0,Y 347.84,Z 307.149,A -85,B 0,C 180,E1 -13696.432,E2 -13696.432} C_VEL
LIN {X 0,Y 347.856,Z 307.152,A -85,B 0,C 180,E1 -13698.86,E2 -13698.86} C_VEL
LIN {X 0,Y 347.764,Z 307.167,A -85,B 0,C 180,E1 -13702.58,E2 -13702.58} C_VEL
LIN {X 0,Y 347.812,Z 307.156,A -85,B 0,C 180,E1 -13705.109,E2 -13705.109} C_VEL
LIN {X 0,Y 347.81,Z 307.156,A -85,B 0,C 180,E1 -13707.694,E2 -13707.694} C_VEL
LIN {X 0,Y 347.765,Z 307.164,A -85,B 0,C 180,E1 -13710.347,E2 -13710.347} C_VEL
LIN {X 0,Y 347.746,Z 307.167,A -85,B 0,C 180,E1 -13714.464,E2 -13714.464} C_VEL
LIN {X 0,Y 347.775,Z 307.161,A -85,B 0,C 180,E1 -13717.989,E2 -13717.989} C_VEL
LIN {X 0,Y 347.752,Z 307.157,A -85,B 0,C 180,E1 -13721.83,E2 -13721.83} C_VEL
LIN {X 0,Y 347.707,Z 307.171,A -85,B 0,C 180,E1 -13725.027,E2 -13725.027} C_VEL
LIN {X 0,Y 347.752,Z 307.166,A -85,B 0,C 180,E1 -13728.397,E2 -13728.397} C_VEL
LIN {X 0,Y 347.775,Z 307.161,A -85,B 0,C 180,E1 -13732.012,E2 -13732.012} C_VEL
LIN {X 0,Y 347.746,Z 307.164,A -85,B 0,C 180,E1 -13735.536,E2 -13735.536} C_VEL
LIN {X 0,Y 347.77,Z 307.197,A -85,B 0,C 180,E1 -13737.561,E2 -13737.561} C_VEL
LIN {X 0,Y 350.677,Z 318.951,A -85,B 0,C 180,E1 -13740.922,E2 -13740.922} C_VEL
LIN {X 0,Y 352.737,Z 329.351,A -85,B 0,C 180,E1 -13743.714,E2 -13743.714} C_VEL
LIN {X 0,Y 352.896,Z 331.806,A -85,B 0,C 180,E1 -13744.332,E2 -13744.332} C_VEL
LIN {X 0,Y 352.105,Z 338.556,A -85,B 0,C 180,E1 -13745.92,E2 -13745.92} C_VEL
LIN {X 0,Y 357.196,Z 363.826,A -85,B 0,C 180,E1 -13746.902,E2 -13746.902} C_VEL
LIN {X 0,Y 359.194,Z 377.094,A -85,B 0,C 180,E1 -13747.349,E2 -13747.349} C_VEL
LIN {X 0,Y 357.657,Z 447.461,A -85,B 0,C 180,E1 -13748.796,E2 -13748.796} C_VEL
LIN {X 0,Y 356.8,Z 460.584,A -85,B 0,C 180,E1 -13749.272,E2 -13749.272} C_VEL
LIN {X 0,Y 355.841,Z 472.646,A -85,B 0,C 180,E1 -13749.93,E2 -13749.93} C_VEL
LIN {X 0,Y 354.684,Z 484.045,A -85,B 0,C 180,E1 -13750.766,E2 -13750.766} C_VEL
LIN {X 0,Y 353.292,Z 494.491,A -85,B 0,C 180,E1 -13751.741,E2 -13751.741} C_VEL
LIN {X 0,Y 351.84,Z 505.236,A -85,B 0,C 180,E1 -13753.014,E2 -13753.014} C_VEL
LIN {X 0,Y 350.388,Z 515.24,A -85,B 0,C 180,E1 -13754.491,E2 -13754.491} C_VEL
LIN {X 0,Y 349.329,Z 523.62,A -85,B 0,C 180,E1 -13756.029,E2 -13756.029} C_VEL
LIN {X 0,Y 348.082,Z 531.272,A -85,B 0,C 180,E1 -13757.76,E2 -13757.76} C_VEL
LIN {X 0,Y 347.281,Z 537.445,A -85,B 0,C 180,E1 -13759.506,E2 -13759.506} C_VEL
LIN {X 0,Y 346.716,Z 542.367,A -85,B 0,C 180,E1 -13761.255,E2 -13761.255} C_VEL
LIN {X 0,Y 346.344,Z 546.179,A -85,B 0,C 180,E1 -13763.006,E2 -13763.006} C_VEL
LIN {X 0,Y 346.231,Z 548.155,A -85,B 0,C 180,E1 -13764.174,E2 -13764.174} C_VEL
LIN {X 0,Y 346.177,Z 549.723,A -85,B 0,C 180,E1 -13765.342,E2 -13765.342} C_VEL
LIN {X 0,Y 346.147,Z 550.851,A -85,B 0,C 180,E1 -13766.508,E2 -13766.508} C_VEL
LIN {X 0,Y 346.161,Z 551.903,A -85,B 0,C 180,E1 -13768.836,E2 -13768.836} C_VEL
LIN {X 0,Y 346.233,Z 551.852,A -85,B 0,C 180,E1 -13770,E2 -13770} C_VEL
LIN {X 0,Y 346.194,Z 551.381,A -85,B 0,C 180,E1 -13771.163,E2 -13771.163} C_VEL
LIN {X 0,Y 346.168,Z 549.194,A -85,B 0,C 180,E1 -13773.491,E2 -13773.491} C_VEL
LIN {X 0,Y 346.199,Z 545.955,A -85,B 0,C 180,E1 -13775.505,E2 -13775.505} C_VEL
LIN {X 0,Y 346.433,Z 541.155,A -85,B 0,C 180,E1 -13777.577,E2 -13777.577} C_VEL
LIN {X 0,Y 346.818,Z 534.785,A -85,B 0,C 180,E1 -13779.623,E2 -13779.623} C_VEL
LIN {X 0,Y 347.384,Z 527.841,A -85,B 0,C 180,E1 -13781.376,E2 -13781.376} C_VEL
LIN {X 0,Y 348.3,Z 519.145,A -85,B 0,C 180,E1 -13783.12,E2 -13783.12} C_VEL
LIN {X 0,Y 349.289,Z 509.198,A -85,B 0,C 180,E1 -13784.718,E2 -13784.718} C_VEL
LIN {X 0,Y 350.097,Z 499.16,A -85,B 0,C 180,E1 -13786.022,E2 -13786.022} C_VEL
LIN {X 0,Y 351.169,Z 487.991,A -85,B 0,C 180,E1 -13787.169,E2 -13787.169} C_VEL
LIN {X 0,Y 352.213,Z 475.453,A -85,B 0,C 180,E1 -13788.166,E2 -13788.166} C_VEL
LIN {X 0,Y 353.061,Z 463.471,A -85,B 0,C 180,E1 -13788.872,E2 -13788.872} C_VEL
LIN {X 0,Y 353.749,Z 450.287,A -85,B 0,C 180,E1 -13789.399,E2 -13789.399} C_VEL
LIN {X 0,Y 354.1,Z 430.593,A -85,B 0,C 180,E1 -13789.851,E2 -13789.851} C_VEL
LIN {X 0,Y 354.947,Z 374.627,A -85,B 0,C 180,E1 -13790.975,E2 -13790.975} C_VEL
LIN {X 0,Y 349.977,Z 339.074,A -85,B 0,C 180,E1 -13791.997,E2 -13791.997} C_VEL
LIN {X 0,Y 351.189,Z 326.6,A -85,B 0,C 180,E1 -13794.85,E2 -13794.85} C_VEL
LIN {X 0,Y 350.997,Z 323.016,A -85,B 0,C 180,E1 -13795.705,E2 -13795.705} C_VEL
LIN {X 0,Y 348.747,Z 311.507,A -85,B 0,C 180,E1 -13798.603,E2 -13798.603} C_VEL
LIN {X 0,Y 347.822,Z 307.16,A -85,B 0,C 180,E1 -13799.762,E2 -13799.762} C_VEL
LIN {X 0,Y 347.748,Z 307.169,A -85,B 0,C 180,E1 -13804.043,E2 -13804.043} C_VEL
LIN {X 0,Y 347.76,Z 307.163,A -85,B 0,C 180,E1 -13807.32,E2 -13807.32} C_VEL
LIN {X 0,Y 347.731,Z 307.172,A -85,B 0,C 180,E1 -13810.296,E2 -13810.296} C_VEL
LIN {X 0,Y 347.721,Z 307.167,A -85,B 0,C 180,E1 -13813.407,E2 -13813.407} C_VEL
LIN {X 0,Y 347.723,Z 307.172,A -85,B 0,C 180,E1 -13816.686,E2 -13816.686} C_VEL
LIN {X 0,Y 347.745,Z 307.166,A -85,B 0,C 180,E1 -13820.172,E2 -13820.172} C_VEL
LIN {X 0,Y 347.759,Z 307.169,A -85,B 0,C 180,E1 -13822.678,E2 -13822.678} C_VEL
LIN {X 0,Y 347.745,Z 307.165,A -85,B 0,C 180,E1 -13825.956,E2 -13825.956} C_VEL
LIN {X 0,Y 347.746,Z 307.165,A -85,B 0,C 180,E1 -13829.651,E2 -13829.651} C_VEL
LIN {X 0,Y 347.827,Z 307.155,A -85,B 0,C 180,E1 -13833.607,E2 -13833.607} C_VEL
LIN {X 0,Y 347.785,Z 307.159,A -85,B 0,C 180,E1 -13836.161,E2 -13836.161} C_VEL
LIN {X 0,Y 347.813,Z 307.156,A -85,B 0,C 180,E1 -13839.909,E2 -13839.909} C_VEL
LIN {X 0,Y 347.862,Z 307.15,A -85,B 0,C 180,E1 -13842.359,E2 -13842.359} C_VEL
LIN {X 0,Y 347.893,Z 307.147,A -85,B 0,C 180,E1 -13845.97,E2 -13845.97} C_VEL
LIN {X 0,Y 347.924,Z 307.148,A -85,B 0,C 180,E1 -13849.525,E2 -13849.525} C_VEL
LIN {X 0,Y 348.088,Z 307.123,A -85,B 0,C 180,E1 -13853.042,E2 -13853.042} C_VEL
LIN {X 0,Y 348.201,Z 307.114,A -85,B 0,C 180,E1 -13857.686,E2 -13857.686} C_VEL
LIN {X 0,Y 348.32,Z 307.096,A -85,B 0,C 180,E1 -13860,E2 -13860} C_VEL
LIN {X 0,Y 348.201,Z 307.109,A -85,B 0,C 180,E1 -13862.313,E2 -13862.313} C_VEL
LIN {X 0,Y 348.065,Z 307.124,A -85,B 0,C 180,E1 -13866.958,E2 -13866.958} C_VEL
LIN {X 0,Y 347.923,Z 307.144,A -85,B 0,C 180,E1 -13870.474,E2 -13870.474} C_VEL
LIN {X 0,Y 347.893,Z 307.152,A -85,B 0,C 180,E1 -13874.15,E2 -13874.15} C_VEL
LIN {X 0,Y 347.886,Z 307.153,A -85,B 0,C 180,E1 -13878.29,E2 -13878.29} C_VEL
LIN {X 0,Y 347.762,Z 307.163,A -85,B 0,C 180,E1 -13881.626,E2 -13881.626} C_VEL
LIN {X 0,Y 347.806,Z 307.157,A -85,B 0,C 180,E1 -13885.109,E2 -13885.109} C_VEL
LIN {X 0,Y 347.806,Z 307.157,A -85,B 0,C 180,E1 -13887.694,E2 -13887.694} C_VEL
LIN {X 0,Y 347.759,Z 307.167,A -85,B 0,C 180,E1 -13890.347,E2 -13890.347} C_VEL
LIN {X 0,Y 347.74,Z 307.169,A -85,B 0,C 180,E1 -13894.464,E2 -13894.464} C_VEL
LIN {X 0,Y 347.768,Z 307.162,A -85,B 0,C 180,E1 -13897.989,E2 -13897.989} C_VEL
LIN {X 0,Y 347.746,Z 307.164,A -85,B 0,C 180,E1 -13901.831,E2 -13901.831} C_VEL
LIN {X 0,Y 347.701,Z 307.176,A -85,B 0,C 180,E1 -13905.027,E2 -13905.027} C_VEL
LIN {X 0,Y 347.737,Z 307.166,A -85,B 0,C 180,E1 -13908.399,E2 -13908.399} C_VEL
LIN {X 0,Y 347.753,Z 307.165,A -85,B 0,C 180,E1 -13912.679,E2 -13912.679} C_VEL
LIN {X 0,Y 347.745,Z 307.165,A -85,B 0,C 180,E1 -13915.957,E2 -13915.957} C_VEL
LIN {X 0,Y 347.735,Z 307.169,A -85,B 0,C 180,E1 -13919.652,E2 -13919.652} C_VEL
LIN {X 0,Y 347.734,Z 307.171,A -85,B 0,C 180,E1 -13923.6,E2 -13923.6} C_VEL
LIN {X 0,Y 347.749,Z 307.165,A -85,B 0,C 180,E1 -13926.16,E2 -13926.16} C_VEL
LIN {X 0,Y 347.798,Z 307.161,A -85,B 0,C 180,E1 -13929.909,E2 -13929.909} C_VEL
LIN {X 0,Y 347.831,Z 307.159,A -85,B 0,C 180,E1 -13933.569,E2 -13933.569} C_VEL
LIN {X 0,Y 347.906,Z 307.162,A -85,B 0,C 180,E1 -13935.911,E2 -13935.911} C_VEL
LIN {X 0,Y 349.427,Z 314.992,A -85,B 0,C 180,E1 -13938.044,E2 -13938.044} C_VEL
LIN {X 0,Y 352.806,Z 325.988,A -85,B 0,C 180,E1 -13938.478,E2 -13938.478} C_VEL
LIN {X 0,Y 355.462,Z 341.354,A -85,B 0,C 180,E1 -13938.944,E2 -13938.944} C_VEL
LIN {X 0,Y 354.034,Z 423.012,A -85,B 0,C 180,E1 -13940.611,E2 -13940.611} C_VEL
LIN {X 0,Y 353.512,Z 436.725,A -85,B 0,C 180,E1 -13941.137,E2 -13941.137} C_VEL
LIN {X 0,Y 352.915,Z 449.03,A -85,B 0,C 180,E1 -13941.843,E2 -13941.843} C_VEL
LIN {X 0,Y 352.057,Z 461.627,A -85,B 0,C 180,E1 -13942.833,E2 -13942.833} C_VEL
LIN {X 0,Y 350.833,Z 472.889,A -85,B 0,C 180,E1 -13943.964,E2 -13943.964} C_VEL
LIN {X 0,Y 349.914,Z 482.979,A -85,B 0,C 180,E1 -13945.248,E2 -13945.248} C_VEL
LIN {X 0,Y 348.961,Z 492.875,A -85,B 0,C 180,E1 -13946.826,E2 -13946.826} C_VEL
LIN {X 0,Y 348.107,Z 501.6,A -85,B 0,C 180,E1 -13948.554,E2 -13948.554} C_VEL
LIN {X 0,Y 347.35,Z 508.59,A -85,B 0,C 180,E1 -13950.29,E2 -13950.29} C_VEL
LIN {X 0,Y 346.846,Z 514.973,A -85,B 0,C 180,E1 -13952.323,E2 -13952.323} C_VEL
LIN {X 0,Y 346.478,Z 519.194,A -85,B 0,C 180,E1 -13954.071,E2 -13954.071} C_VEL
LIN {X 0,Y 346.417,Z 522.967,A -85,B 0,C 180,E1 -13956.231,E2 -13956.231} C_VEL
LIN {X 0,Y 346.15,Z 525.089,A -85,B 0,C 180,E1 -13958.171,E2 -13958.171} C_VEL
LIN {X 0,Y 346.053,Z 526.151,A -85,B 0,C 180,E1 -13960.532,E2 -13960.532} C_VEL
LIN {X 0,Y 346.149,Z 526.099,A -85,B 0,C 180,E1 -13961.715,E2 -13961.715} C_VEL
LIN {X 0,Y 346.306,Z 525.513,A -85,B 0,C 180,E1 -13963.064,E2 -13963.064} C_VEL
LIN {X 0,Y 346.545,Z 523.416,A -85,B 0,C 180,E1 -13965.287,E2 -13965.287} C_VEL
LIN {X 0,Y 346.973,Z 520.62,A -85,B 0,C 180,E1 -13967.08,E2 -13967.08} C_VEL
LIN {X 0,Y 347.53,Z 516.753,A -85,B 0,C 180,E1 -13968.879,E2 -13968.879} C_VEL
LIN {X 0,Y 348.338,Z 511.698,A -85,B 0,C 180,E1 -13970.676,E2 -13970.676} C_VEL
LIN {X 0,Y 349.31,Z 505.28,A -85,B 0,C 180,E1 -13972.475,E2 -13972.475} C_VEL
LIN {X 0,Y 350.583,Z 497.162,A -85,B 0,C 180,E1 -13974.265,E2 -13974.265} C_VEL
LIN {X 0,Y 351.837,Z 488.826,A -85,B 0,C 180,E1 -13975.751,E2 -13975.751} C_VEL
LIN {X 0,Y 353.106,Z 479.797,A -85,B 0,C 180,E1 -13977.068,E2 -13977.068} C_VEL
LIN {X 0,Y 354.42,Z 469.753,A -85,B 0,C 180,E1 -13978.257,E2 -13978.257} C_VEL
LIN {X 0,Y 355.61,Z 458.884,A -85,B 0,C 180,E1 -13979.284,E2 -13979.284} C_VEL
LIN {X 0,Y 356.67,Z 446.84,A -85,B 0,C 180,E1 -13980.163,E2 -13980.163} C_VEL
LIN {X 0,Y 356.93,Z 442.233,A -85,B 0,C 180,E1 -13980.442,E2 -13980.442} C_VEL
LIN {X 0,Y 356.477,Z 438.546,A -85,B 0,C 180,E1 -13980.693,E2 -13980.693} C_VEL
LIN {X 0,Y 351.809,Z 427.078,A -85,B 0,C 180,E1 -13981.573,E2 -13981.573} C_VEL
LIN {X 0,Y 351.429,Z 423.27,A -85,B 0,C 180,E1 -13981.734,E2 -13981.734} C_VEL
LIN {X 0,Y 353.443,Z 344.28,A -85,B 0,C 180,E1 -13983.369,E2 -13983.369} C_VEL
LIN {X 0,Y 351.407,Z 335.852,A -85,B 0,C 180,E1 -13983.729,E2 -13983.729} C_VEL
LIN {X 0,Y 343.538,Z 318.04,A -85,B 0,C 180,E1 -13984.829,E2 -13984.829} C_VEL
LIN {X 0,Y 342.589,Z 315.657,A -85,B 0,C 180,E1 -13984.997,E2 -13984.997} C_VEL
LIN {X 0,Y 340.725,Z 308.033,A -85,B 0,C 180,E1 -13987.387,E2 -13987.387} C_VEL
LIN {X 0,Y 340.685,Z 308.048,A -85,B 0,C 180,E1 -13991.31,E2 -13991.31} C_VEL
LIN {X 0,Y 340.64,Z 308.051,A -85,B 0,C 180,E1 -13994.546,E2 -13994.546} C_VEL
LIN {X 0,Y 340.698,Z 308.044,A -85,B 0,C 180,E1 -13997.955,E2 -13997.955} C_VEL
LIN {X 0,Y 340.732,Z 308.036,A -85,B 0,C 180,E1 -14001.773,E2 -14001.773} C_VEL
LIN {X 0,Y 340.722,Z 308.037,A -85,B 0,C 180,E1 -14005.596,E2 -14005.596} C_VEL
LIN {X 0,Y 340.703,Z 308.035,A -85,B 0,C 180,E1 -14008.956,E2 -14008.956} C_VEL
LIN {X 0,Y 340.777,Z 308.025,A -85,B 0,C 180,E1 -14012.475,E2 -14012.475} C_VEL
LIN {X 0,Y 340.754,Z 308.03,A -85,B 0,C 180,E1 -14015.638,E2 -14015.638} C_VEL
LIN {X 0,Y 340.735,Z 308.036,A -85,B 0,C 180,E1 -14019.474,E2 -14019.474} C_VEL
LIN {X 0,Y 340.858,Z 308.025,A -85,B 0,C 180,E1 -14021.984,E2 -14021.984} C_VEL
LIN {X 0,Y 340.869,Z 308.022,A -85,B 0,C 180,E1 -14025.705,E2 -14025.705} C_VEL
LIN {X 0,Y 340.87,Z 308.017,A -85,B 0,C 180,E1 -14029.306,E2 -14029.306} C_VEL
LIN {X 0,Y 341.074,Z 307.993,A -85,B 0,C 180,E1 -14032.898,E2 -14032.898} C_VEL
LIN {X 0,Y 341.168,Z 307.981,A -85,B 0,C 180,E1 -14037.639,E2 -14037.639} C_VEL
LIN {X 0,Y 341.276,Z 307.974,A -85,B 0,C 180,E1 -14040,E2 -14040} C_VEL
LIN {X 0,Y 341.168,Z 307.978,A -85,B 0,C 180,E1 -14042.361,E2 -14042.361} C_VEL
LIN {X 0,Y 341.075,Z 307.986,A -85,B 0,C 180,E1 -14047.102,E2 -14047.102} C_VEL
LIN {X 0,Y 340.871,Z 308.017,A -85,B 0,C 180,E1 -14050.694,E2 -14050.694} C_VEL
LIN {X 0,Y 340.864,Z 308.026,A -85,B 0,C 180,E1 -14054.325,E2 -14054.325} C_VEL
LIN {X 0,Y 340.839,Z 308.029,A -85,B 0,C 180,E1 -14058.467,E2 -14058.467} C_VEL
LIN {X 0,Y 340.718,Z 308.039,A -85,B 0,C 180,E1 -14061.842,E2 -14061.842} C_VEL
LIN {X 0,Y 340.773,Z 308.033,A -85,B 0,C 180,E1 -14065.665,E2 -14065.665} C_VEL
LIN {X 0,Y 340.741,Z 308.036,A -85,B 0,C 180,E1 -14068.32,E2 -14068.32} C_VEL
LIN {X 0,Y 340.705,Z 308.045,A -85,B 0,C 180,E1 -14071.044,E2 -14071.044} C_VEL
LIN {X 0,Y 340.719,Z 308.039,A -85,B 0,C 180,E1 -14075.279,E2 -14075.279} C_VEL
LIN {X 0,Y 340.711,Z 308.041,A -85,B 0,C 180,E1 -14078.386,E2 -14078.386} C_VEL
LIN {X 0,Y 340.7,Z 308.039,A -85,B 0,C 180,E1 -14082.046,E2 -14082.046} C_VEL
LIN {X 0,Y 340.653,Z 308.05,A -85,B 0,C 180,E1 -14086.227,E2 -14086.227} C_VEL
LIN {X 0,Y 340.69,Z 308.049,A -85,B 0,C 180,E1 -14089.753,E2 -14089.753} C_VEL
LIN {X 0,Y 340.707,Z 308.039,A -85,B 0,C 180,E1 -14093.259,E2 -14093.259} C_VEL
LIN {X 0,Y 340.718,Z 308.142,A -85,B 0,C 180,E1 -14097.042,E2 -14097.042} C_VEL
LIN {X 0,Y 343.767,Z 320.304,A -85,B 0,C 180,E1 -14100.616,E2 -14100.616} C_VEL
LIN {X 0,Y 345.94,Z 331.297,A -85,B 0,C 180,E1 -14103.635,E2 -14103.635} C_VEL
LIN {X 0,Y 345.885,Z 334.434,A -85,B 0,C 180,E1 -14104.419,E2 -14104.419} C_VEL
LIN {X 0,Y 345.469,Z 338.567,A -85,B 0,C 180,E1 -14105.355,E2 -14105.355} C_VEL
LIN {X 0,Y 350.286,Z 361.904,A -85,B 0,C 180,E1 -14106.3,E2 -14106.3} C_VEL
LIN {X 0,Y 352.799,Z 377.476,A -85,B 0,C 180,E1 -14106.855,E2 -14106.855} C_VEL
LIN {X 0,Y 351.212,Z 447.054,A -85,B 0,C 180,E1 -14108.31,E2 -14108.31} C_VEL
LIN {X 0,Y 350.36,Z 460.212,A -85,B 0,C 180,E1 -14108.795,E2 -14108.795} C_VEL
LIN {X 0,Y 349.333,Z 472.299,A -85,B 0,C 180,E1 -14109.463,E2 -14109.463} C_VEL
LIN {X 0,Y 348.012,Z 484.534,A -85,B 0,C 180,E1 -14110.382,E2 -14110.382} C_VEL
LIN {X 0,Y 346.578,Z 494.817,A -85,B 0,C 180,E1 -14111.374,E2 -14111.374} C_VEL
LIN {X 0,Y 345.069,Z 505.461,A -85,B 0,C 180,E1 -14112.67,E2 -14112.67} C_VEL
LIN {X 0,Y 343.464,Z 515.956,A -85,B 0,C 180,E1 -14114.271,E2 -14114.271} C_VEL
LIN {X 0,Y 342.2,Z 525.032,A -85,B 0,C 180,E1 -14116.035,E2 -14116.035} C_VEL
LIN {X 0,Y 340.982,Z 532.381,A -85,B 0,C 180,E1 -14117.803,E2 -14117.803} C_VEL
LIN {X 0,Y 340.039,Z 539.16,A -85,B 0,C 180,E1 -14119.881,E2 -14119.881} C_VEL
LIN {X 0,Y 339.528,Z 543.656,A -85,B 0,C 180,E1 -14121.668,E2 -14121.668} C_VEL
LIN {X 0,Y 339.275,Z 546.035,A -85,B 0,C 180,E1 -14122.86,E2 -14122.86} C_VEL
LIN {X 0,Y 339.137,Z 548.078,A -85,B 0,C 180,E1 -14124.109,E2 -14124.109} C_VEL
LIN {X 0,Y 339.08,Z 549.535,A -85,B 0,C 180,E1 -14125.244,E2 -14125.244} C_VEL
LIN {X 0,Y 339.072,Z 550.631,A -85,B 0,C 180,E1 -14126.435,E2 -14126.435} C_VEL
LIN {X 0,Y 339.063,Z 551.646,A -85,B 0,C 180,E1 -14128.812,E2 -14128.812} C_VEL
LIN {X 0,Y 339.138,Z 551.577,A -85,B 0,C 180,E1 -14130,E2 -14130} C_VEL
LIN {X 0,Y 339.096,Z 551.072,A -85,B 0,C 180,E1 -14131.187,E2 -14131.187} C_VEL
LIN {X 0,Y 339.094,Z 548.849,A -85,B 0,C 180,E1 -14133.564,E2 -14133.564} C_VEL
LIN {X 0,Y 339.101,Z 545.899,A -85,B 0,C 180,E1 -14135.438,E2 -14135.438} C_VEL
LIN {X 0,Y 339.268,Z 542.226,A -85,B 0,C 180,E1 -14137.139,E2 -14137.139} C_VEL
LIN {X 0,Y 339.57,Z 537.25,A -85,B 0,C 180,E1 -14138.929,E2 -14138.929} C_VEL
LIN {X 0,Y 340.026,Z 530.977,A -85,B 0,C 180,E1 -14140.72,E2 -14140.72} C_VEL
LIN {X 0,Y 340.822,Z 523.139,A -85,B 0,C 180,E1 -14142.504,E2 -14142.504} C_VEL
LIN {X 0,Y 341.653,Z 515.114,A -85,B 0,C 180,E1 -14143.987,E2 -14143.987} C_VEL
LIN {X 0,Y 342.576,Z 505.301,A -85,B 0,C 180,E1 -14145.467,E2 -14145.467} C_VEL
LIN {X 0,Y 343.608,Z 494.387,A -85,B 0,C 180,E1 -14146.792,E2 -14146.792} C_VEL
LIN {X 0,Y 344.671,Z 483.734,A -85,B 0,C 180,E1 -14147.809,E2 -14147.809} C_VEL
LIN {X 0,Y 345.643,Z 470.866,A -85,B 0,C 180,E1 -14148.754,E2 -14148.754} C_VEL
LIN {X 0,Y 346.542,Z 457.947,A -85,B 0,C 180,E1 -14149.434,E2 -14149.434} C_VEL
LIN {X 0,Y 347.099,Z 445.224,A -85,B 0,C 180,E1 -14149.863,E2 -14149.863} C_VEL
LIN {X 0,Y 348.203,Z 375.619,A -85,B 0,C 180,E1 -14151.303,E2 -14151.303} C_VEL
LIN {X 0,Y 343.101,Z 338.834,A -85,B 0,C 180,E1 -14152.379,E2 -14152.379} C_VEL
LIN {X 0,Y 344.263,Z 325.988,A -85,B 0,C 180,E1 -14155.385,E2 -14155.385} C_VEL
LIN {X 0,Y 342.276,Z 315.021,A -85,B 0,C 180,E1 -14158.181,E2 -14158.181} C_VEL
LIN {X 0,Y 340.758,Z 308.042,A -85,B 0,C 180,E1 -14160.078,E2 -14160.078} C_VEL
LIN {X 0,Y 340.722,Z 308.044,A -85,B 0,C 180,E1 -14164.404,E2 -14164.404} C_VEL
LIN {X 0,Y 340.709,Z 308.047,A -85,B 0,C 180,E1 -14168.385,E2 -14168.385} C_VEL
LIN {X 0,Y 340.697,Z 308.045,A -85,B 0,C 180,E1 -14172.045,E2 -14172.045} C_VEL
LIN {X 0,Y 340.65,Z 308.052,A -85,B 0,C 180,E1 -14176.226,E2 -14176.226} C_VEL
LIN {X 0,Y 340.686,Z 308.044,A -85,B 0,C 180,E1 -14179.752,E2 -14179.752} C_VEL
LIN {X 0,Y 340.702,Z 308.044,A -85,B 0,C 180,E1 -14183.258,E2 -14183.258} C_VEL
LIN {X 0,Y 340.689,Z 308.044,A -85,B 0,C 180,E1 -14186.153,E2 -14186.153} C_VEL
LIN {X 0,Y 340.738,Z 308.039,A -85,B 0,C 180,E1 -14190.329,E2 -14190.329} C_VEL
LIN {X 0,Y 340.8,Z 308.036,A -85,B 0,C 180,E1 -14193.019,E2 -14193.019} C_VEL
LIN {X 0,Y 340.752,Z 308.037,A -85,B 0,C 180,E1 -14195.638,E2 -14195.638} C_VEL
LIN {X 0,Y 340.744,Z 308.04,A -85,B 0,C 180,E1 -14199.474,E2 -14199.474} C_VEL
LIN {X 0,Y 340.854,Z 308.023,A -85,B 0,C 180,E1 -14201.984,E2 -14201.984} C_VEL
LIN {X 0,Y 340.865,Z 308.024,A -85,B 0,C 180,E1 -14205.705,E2 -14205.705} C_VEL
LIN {X 0,Y 340.866,Z 308.025,A -85,B 0,C 180,E1 -14209.306,E2 -14209.306} C_VEL
LIN {X 0,Y 341.056,Z 307.999,A -85,B 0,C 180,E1 -14212.898,E2 -14212.898} C_VEL
LIN {X 0,Y 341.163,Z 307.99,A -85,B 0,C 180,E1 -14217.638,E2 -14217.638} C_VEL
LIN {X 0,Y 341.271,Z 307.974,A -85,B 0,C 180,E1 -14220,E2 -14220} C_VEL
LIN {X 0,Y 341.163,Z 307.985,A -85,B 0,C 180,E1 -14222.361,E2 -14222.361} C_VEL
LIN {X 0,Y 341.013,Z 308.003,A -85,B 0,C 180,E1 -14227.103,E2 -14227.103} C_VEL
LIN {X 0,Y 340.866,Z 308.021,A -85,B 0,C 180,E1 -14230.694,E2 -14230.694} C_VEL
LIN {X 0,Y 340.858,Z 308.027,A -85,B 0,C 180,E1 -14234.325,E2 -14234.325} C_VEL
LIN {X 0,Y 340.832,Z 308.029,A -85,B 0,C 180,E1 -14238.466,E2 -14238.466} C_VEL
LIN {X 0,Y 340.713,Z 308.041,A -85,B 0,C 180,E1 -14241.842,E2 -14241.842} C_VEL
LIN {X 0,Y 340.767,Z 308.034,A -85,B 0,C 180,E1 -14245.665,E2 -14245.665} C_VEL
LIN {X 0,Y 340.736,Z 308.042,A -85,B 0,C 180,E1 -14248.32,E2 -14248.32} C_VEL
LIN {X 0,Y 340.699,Z 308.043,A -85,B 0,C 180,E1 -14251.044,E2 -14251.044} C_VEL
LIN {X 0,Y 340.713,Z 308.041,A -85,B 0,C 180,E1 -14255.279,E2 -14255.279} C_VEL
LIN {X 0,Y 340.705,Z 308.043,A -85,B 0,C 180,E1 -14258.386,E2 -14258.386} C_VEL
LIN {X 0,Y 340.694,Z 308.043,A -85,B 0,C 180,E1 -14262.046,E2 -14262.046} C_VEL
LIN {X 0,Y 340.647,Z 308.048,A -85,B 0,C 180,E1 -14266.228,E2 -14266.228} C_VEL
LIN {X 0,Y 340.667,Z 308.049,A -85,B 0,C 180,E1 -14268.689,E2 -14268.689} C_VEL
LIN {X 0,Y 340.715,Z 308.041,A -85,B 0,C 180,E1 -14271.771,E2 -14271.771} C_VEL
LIN {X 0,Y 340.72,Z 308.042,A -85,B 0,C 180,E1 -14275.596,E2 -14275.596} C_VEL
LIN {X 0,Y 340.69,Z 308.046,A -85,B 0,C 180,E1 -14278.955,E2 -14278.955} C_VEL
LIN {X 0,Y 340.708,Z 308.043,A -85,B 0,C 180,E1 -14283.012,E2 -14283.012} C_VEL
LIN {X 0,Y 340.703,Z 308.043,A -85,B 0,C 180,E1 -14286.926,E2 -14286.926} C_VEL
LIN {X 0,Y 340.757,Z 308.035,A -85,B 0,C 180,E1 -14290.732,E2 -14290.732} C_VEL
LIN {X 0,Y 340.816,Z 308.031,A -85,B 0,C 180,E1 -14294.451,E2 -14294.451} C_VEL
LIN {X 0,Y 340.864,Z 308.208,A -85,B 0,C 180,E1 -14295.676,E2 -14295.676} C_VEL
LIN {X 0,Y 342.312,Z 315.266,A -85,B 0,C 180,E1 -14297.643,E2 -14297.643} C_VEL
LIN {X 0,Y 346.334,Z 328.383,A -85,B 0,C 180,E1 -14298.17,E2 -14298.17} C_VEL
LIN {X 0,Y 348.714,Z 342.513,A -85,B 0,C 180,E1 -14298.605,E2 -14298.605} C_VEL
LIN {X 0,Y 347.247,Z 423.055,A -85,B 0,C 180,E1 -14300.278,E2 -14300.278} C_VEL
LIN {X 0,Y 346.743,Z 436.085,A -85,B 0,C 180,E1 -14300.779,E2 -14300.779} C_VEL
LIN {X 0,Y 346.077,Z 449.191,A -85,B 0,C 180,E1 -14301.534,E2 -14301.534} C_VEL
LIN {X 0,Y 345.318,Z 460.243,A -85,B 0,C 180,E1 -14302.399,E2 -14302.399} C_VEL
LIN {X 0,Y 344.321,Z 469.214,A -85,B 0,C 180,E1 -14303.26,E2 -14303.26} C_VEL
LIN {X 0,Y 343.349,Z 480.019,A -85,B 0,C 180,E1 -14304.568,E2 -14304.568} C_VEL
LIN {X 0,Y 342.394,Z 488.855,A -85,B 0,C 180,E1 -14305.881,E2 -14305.881} C_VEL
LIN {X 0,Y 341.445,Z 498.438,A -85,B 0,C 180,E1 -14307.641,E2 -14307.641} C_VEL
LIN {X 0,Y 340.585,Z 506.091,A -85,B 0,C 180,E1 -14309.409,E2 -14309.409} C_VEL
LIN {X 0,Y 340.029,Z 512.228,A -85,B 0,C 180,E1 -14311.185,E2 -14311.185} C_VEL
LIN {X 0,Y 339.616,Z 517.111,A -85,B 0,C 180,E1 -14312.966,E2 -14312.966} C_VEL
LIN {X 0,Y 339.405,Z 520.878,A -85,B 0,C 180,E1 -14314.751,E2 -14314.751} C_VEL
LIN {X 0,Y 339.336,Z 523.221,A -85,B 0,C 180,E1 -14316.213,E2 -14316.213} C_VEL
LIN {X 0,Y 339.032,Z 525.451,A -85,B 0,C 180,E1 -14318.344,E2 -14318.344} C_VEL
LIN {X 0,Y 338.986,Z 526.437,A -85,B 0,C 180,E1 -14320.754,E2 -14320.754} C_VEL
LIN {X 0,Y 339.071,Z 526.337,A -85,B 0,C 180,E1 -14321.963,E2 -14321.963} C_VEL
LIN {X 0,Y 339.241,Z 525.793,A -85,B 0,C 180,E1 -14323.173,E2 -14323.173} C_VEL
LIN {X 0,Y 339.32,Z 524.853,A -85,B 0,C 180,E1 -14324.392,E2 -14324.392} C_VEL
LIN {X 0,Y 339.54,Z 523.508,A -85,B 0,C 180,E1 -14325.61,E2 -14325.61} C_VEL
LIN {X 0,Y 339.993,Z 520.63,A -85,B 0,C 180,E1 -14327.442,E2 -14327.442} C_VEL
LIN {X 0,Y 340.614,Z 516.674,A -85,B 0,C 180,E1 -14329.277,E2 -14329.277} C_VEL
LIN {X 0,Y 341.671,Z 510.506,A -85,B 0,C 180,E1 -14331.415,E2 -14331.415} C_VEL
LIN {X 0,Y 342.728,Z 503.691,A -85,B 0,C 180,E1 -14333.25,E2 -14333.25} C_VEL
LIN {X 0,Y 344.161,Z 495.165,A -85,B 0,C 180,E1 -14335.07,E2 -14335.07} C_VEL
LIN {X 0,Y 345.695,Z 485.292,A -85,B 0,C 180,E1 -14336.731,E2 -14336.731} C_VEL
LIN {X 0,Y 347.116,Z 475.296,A -85,B 0,C 180,E1 -14338.082,E2 -14338.082} C_VEL
LIN {X 0,Y 348.483,Z 464.323,A -85,B 0,C 180,E1 -14339.266,E2 -14339.266} C_VEL
LIN {X 0,Y 349.612,Z 453.457,A -85,B 0,C 180,E1 -14340.186,E2 -14340.186} C_VEL
LIN {X 0,Y 350.565,Z 440.941,A -85,B 0,C 180,E1 -14340.995,E2 -14340.995} C_VEL
LIN {X 0,Y 351.188,Z 428.074,A -85,B 0,C 180,E1 -14341.584,E2 -14341.584} C_VEL
LIN {X 0,Y 351.429,Z 423.27,A -85,B 0,C 180,E1 -14341.734,E2 -14341.734} C_VEL
LIN {X 0,Y 351.182,Z 417.499,A -85,B 0,C 180,E1 -14341.932,E2 -14341.932} C_VEL
LIN {X 0,Y 348.831,Z 408.183,A -85,B 0,C 180,E1 -14342.34,E2 -14342.34} C_VEL
LIN {X 0,Y 346.341,Z 398.838,A -85,B 0,C 180,E1 -14342.729,E2 -14342.729} C_VEL
LIN {X 0,Y 345.873,Z 393.016,A -85,B 0,C 180,E1 -14342.892,E2 -14342.892} C_VEL
LIN {X 0,Y 347.096,Z 345.173,A -85,B 0,C 180,E1 -14343.884,E2 -14343.884} C_VEL
LIN {X 0,Y 345.405,Z 338.555,A -85,B 0,C 180,E1 -14344.184,E2 -14344.184} C_VEL
LIN {X 0,Y 337.047,Z 319.442,A -85,B 0,C 180,E1 -14345.398,E2 -14345.398} C_VEL
LIN {X 0,Y 335.395,Z 315.905,A -85,B 0,C 180,E1 -14345.682,E2 -14345.682} C_VEL
LIN {X 0,Y 333.68,Z 308.911,A -85,B 0,C 180,E1 -14347.934,E2 -14347.934} C_VEL
LIN {X 0,Y 333.646,Z 308.927,A -85,B 0,C 180,E1 -14350.768,E2 -14350.768} C_VEL
LIN {X 0,Y 333.593,Z 308.928,A -85,B 0,C 180,E1 -14354.251,E2 -14354.251} C_VEL
LIN {X 0,Y 333.641,Z 308.923,A -85,B 0,C 180,E1 -14357.619,E2 -14357.619} C_VEL
LIN {X 0,Y 333.652,Z 308.921,A -85,B 0,C 180,E1 -14361.202,E2 -14361.202} C_VEL
LIN {X 0,Y 333.675,Z 308.915,A -85,B 0,C 180,E1 -14363.861,E2 -14363.861} C_VEL
LIN {X 0,Y 333.643,Z 308.919,A -85,B 0,C 180,E1 -14367.413,E2 -14367.413} C_VEL
LIN {X 0,Y 333.71,Z 308.913,A -85,B 0,C 180,E1 -14371.028,E2 -14371.028} C_VEL
LIN {X 0,Y 333.735,Z 308.908,A -85,B 0,C 180,E1 -14373.754,E2 -14373.754} C_VEL
LIN {X 0,Y 333.657,Z 308.92,A -85,B 0,C 180,E1 -14377.72,E2 -14377.72} C_VEL
LIN {X 0,Y 333.794,Z 308.902,A -85,B 0,C 180,E1 -14381.59,E2 -14381.59} C_VEL
LIN {X 0,Y 333.808,Z 308.899,A -85,B 0,C 180,E1 -14385.577,E2 -14385.577} C_VEL
LIN {X 0,Y 333.833,Z 308.894,A -85,B 0,C 180,E1 -14389.078,E2 -14389.078} C_VEL
LIN {X 0,Y 334.024,Z 308.871,A -85,B 0,C 180,E1 -14392.748,E2 -14392.748} C_VEL
LIN {X 0,Y 333.809,Z 308.9,A -85,B 0,C 180,E1 -14395.169,E2 -14395.169} C_VEL
LIN {X 0,Y 334.105,Z 308.861,A -85,B 0,C 180,E1 -14397.589,E2 -14397.589} C_VEL
LIN {X 0,Y 334.227,Z 308.852,A -85,B 0,C 180,E1 -14400,E2 -14400} C_VEL
LIN {X 0,Y 334.105,Z 308.858,A -85,B 0,C 180,E1 -14402.411,E2 -14402.411} C_VEL
LIN {X 0,Y 334.025,Z 308.864,A -85,B 0,C 180,E1 -14407.253,E2 -14407.253} C_VEL
LIN {X 0,Y 333.834,Z 308.891,A -85,B 0,C 180,E1 -14410.922,E2 -14410.922} C_VEL
LIN {X 0,Y 333.809,Z 308.901,A -85,B 0,C 180,E1 -14414.635,E2 -14414.635} C_VEL
LIN {X 0,Y 333.798,Z 308.905,A -85,B 0,C 180,E1 -14418.656,E2 -14418.656} C_VEL
LIN {X 0,Y 333.657,Z 308.921,A -85,B 0,C 180,E1 -14422.281,E2 -14422.281} C_VEL
LIN {X 0,Y 333.736,Z 308.911,A -85,B 0,C 180,E1 -14426.247,E2 -14426.247} C_VEL
LIN {X 0,Y 333.711,Z 308.911,A -85,B 0,C 180,E1 -14428.972,E2 -14428.972} C_VEL
LIN {X 0,Y 333.644,Z 308.918,A -85,B 0,C 180,E1 -14432.587,E2 -14432.587} C_VEL
LIN {X 0,Y 333.677,Z 308.913,A -85,B 0,C 180,E1 -14436.139,E2 -14436.139} C_VEL
LIN {X 0,Y 333.648,Z 308.91,A -85,B 0,C 180,E1 -14439.193,E2 -14439.193} C_VEL
LIN {X 0,Y 333.634,Z 308.923,A -85,B 0,C 180,E1 -14442.5,E2 -14442.5} C_VEL
LIN {X 0,Y 333.598,Z 308.93,A -85,B 0,C 180,E1 -14445.955,E2 -14445.955} C_VEL
LIN {X 0,Y 333.649,Z 308.924,A -85,B 0,C 180,E1 -14449.316,E2 -14449.316} C_VEL
LIN {X 0,Y 333.667,Z 308.915,A -85,B 0,C 180,E1 -14453.168,E2 -14453.168} C_VEL
LIN {X 0,Y 333.672,Z 309.031,A -85,B 0,C 180,E1 -14456.479,E2 -14456.479} C_VEL
LIN {X 0,Y 336.484,Z 320.377,A -85,B 0,C 180,E1 -14459.915,E2 -14459.915} C_VEL
LIN {X 0,Y 338.881,Z 331.571,A -85,B 0,C 180,E1 -14463.097,E2 -14463.097} C_VEL
LIN {X 0,Y 339.204,Z 334.669,A -85,B 0,C 180,E1 -14463.925,E2 -14463.925} C_VEL
LIN {X 0,Y 338.744,Z 337.908,A -85,B 0,C 180,E1 -14464.715,E2 -14464.715} C_VEL
LIN {X 0,Y 343.898,Z 362.611,A -85,B 0,C 180,E1 -14465.775,E2 -14465.775} C_VEL
LIN {X 0,Y 346.402,Z 377.845,A -85,B 0,C 180,E1 -14466.339,E2 -14466.339} C_VEL
LIN {X 0,Y 344.785,Z 446.724,A -85,B 0,C 180,E1 -14467.806,E2 -14467.806} C_VEL
LIN {X 0,Y 343.911,Z 459.901,A -85,B 0,C 180,E1 -14468.299,E2 -14468.299} C_VEL
LIN {X 0,Y 342.804,Z 472.004,A -85,B 0,C 180,E1 -14468.975,E2 -14468.975} C_VEL
LIN {X 0,Y 341.564,Z 483.421,A -85,B 0,C 180,E1 -14469.84,E2 -14469.84} C_VEL
LIN {X 0,Y 339.877,Z 495.171,A -85,B 0,C 180,E1 -14470.993,E2 -14470.993} C_VEL
LIN {X 0,Y 338.29,Z 505.704,A -85,B 0,C 180,E1 -14472.312,E2 -14472.312} C_VEL
LIN {X 0,Y 336.796,Z 514.796,A -85,B 0,C 180,E1 -14473.719,E2 -14473.719} C_VEL
LIN {X 0,Y 335.521,Z 523.726,A -85,B 0,C 180,E1 -14475.442,E2 -14475.442} C_VEL
LIN {X 0,Y 334.188,Z 531.253,A -85,B 0,C 180,E1 -14477.243,E2 -14477.243} C_VEL
LIN {X 0,Y 333.282,Z 537.328,A -85,B 0,C 180,E1 -14479.059,E2 -14479.059} C_VEL
LIN {X 0,Y 332.627,Z 542.162,A -85,B 0,C 180,E1 -14480.882,E2 -14480.882} C_VEL
LIN {X 0,Y 332.202,Z 545.891,A -85,B 0,C 180,E1 -14482.707,E2 -14482.707} C_VEL
LIN {X 0,Y 332.032,Z 548.184,A -85,B 0,C 180,E1 -14484.176,E2 -14484.176} C_VEL
LIN {X 0,Y 331.997,Z 550.412,A -85,B 0,C 180,E1 -14486.358,E2 -14486.358} C_VEL
LIN {X 0,Y 331.966,Z 551.391,A -85,B 0,C 180,E1 -14488.786,E2 -14488.786} C_VEL
LIN {X 0,Y 332.043,Z 551.296,A -85,B 0,C 180,E1 -14490,E2 -14490} C_VEL
LIN {X 0,Y 331.999,Z 550.761,A -85,B 0,C 180,E1 -14491.213,E2 -14491.213} C_VEL
LIN {X 0,Y 332.019,Z 548.501,A -85,B 0,C 180,E1 -14493.64,E2 -14493.64} C_VEL
LIN {X 0,Y 332.018,Z 546.744,A -85,B 0,C 180,E1 -14494.857,E2 -14494.857} C_VEL
LIN {X 0,Y 332.157,Z 543.233,A -85,B 0,C 180,E1 -14496.682,E2 -14496.682} C_VEL
LIN {X 0,Y 332.38,Z 538.604,A -85,B 0,C 180,E1 -14498.511,E2 -14498.511} C_VEL
LIN {X 0,Y 332.932,Z 531.584,A -85,B 0,C 180,E1 -14500.644,E2 -14500.644} C_VEL
LIN {X 0,Y 333.715,Z 523.981,A -85,B 0,C 180,E1 -14502.466,E2 -14502.466} C_VEL
LIN {X 0,Y 334.511,Z 516.204,A -85,B 0,C 180,E1 -14503.981,E2 -14503.981} C_VEL
LIN {X 0,Y 335.365,Z 508.426,A -85,B 0,C 180,E1 -14505.238,E2 -14505.238} C_VEL
LIN {X 0,Y 336.208,Z 498.72,A -85,B 0,C 180,E1 -14506.547,E2 -14506.547} C_VEL
LIN {X 0,Y 337.349,Z 487.576,A -85,B 0,C 180,E1 -14507.738,E2 -14507.738} C_VEL
LIN {X 0,Y 338.498,Z 475.075,A -85,B 0,C 180,E1 -14508.772,E2 -14508.772} C_VEL
LIN {X 0,Y 339.409,Z 463.158,A -85,B 0,C 180,E1 -14509.505,E2 -14509.505} C_VEL
LIN {X 0,Y 340.137,Z 450.102,A -85,B 0,C 180,E1 -14510.051,E2 -14510.051} C_VEL
LIN {X 0,Y 340.489,Z 431.492,A -85,B 0,C 180,E1 -14510.502,E2 -14510.502} C_VEL
LIN {X 0,Y 341.431,Z 376.314,A -85,B 0,C 180,E1 -14511.651,E2 -14511.651} C_VEL
LIN {X 0,Y 336.21,Z 338.478,A -85,B 0,C 180,E1 -14512.804,E2 -14512.804} C_VEL
LIN {X 0,Y 337.285,Z 328.067,A -85,B 0,C 180,E1 -14515.287,E2 -14515.287} C_VEL
LIN {X 0,Y 336.252,Z 321.176,A -85,B 0,C 180,E1 -14517.054,E2 -14517.054} C_VEL
LIN {X 0,Y 334.009,Z 310.324,A -85,B 0,C 180,E1 -14519.947,E2 -14519.947} C_VEL
LIN {X 0,Y 333.698,Z 308.921,A -85,B 0,C 180,E1 -14520.361,E2 -14520.361} C_VEL
LIN {X 0,Y 333.685,Z 308.918,A -85,B 0,C 180,E1 -14524.773,E2 -14524.773} C_VEL
LIN {X 0,Y 333.651,Z 308.921,A -85,B 0,C 180,E1 -14527.65,E2 -14527.65} C_VEL
LIN {X 0,Y 333.645,Z 308.924,A -85,B 0,C 180,E1 -14530.767,E2 -14530.767} C_VEL
LIN {X 0,Y 333.591,Z 308.932,A -85,B 0,C 180,E1 -14534.25,E2 -14534.25} C_VEL
LIN {X 0,Y 333.639,Z 308.922,A -85,B 0,C 180,E1 -14537.618,E2 -14537.618} C_VEL
LIN {X 0,Y 333.65,Z 308.922,A -85,B 0,C 180,E1 -14541.201,E2 -14541.201} C_VEL
LIN {X 0,Y 333.673,Z 308.918,A -85,B 0,C 180,E1 -14543.86,E2 -14543.86} C_VEL
LIN {X 0,Y 333.64,Z 308.923,A -85,B 0,C 180,E1 -14547.412,E2 -14547.412} C_VEL
LIN {X 0,Y 333.687,Z 308.921,A -85,B 0,C 180,E1 -14551.025,E2 -14551.025} C_VEL
LIN {X 0,Y 333.731,Z 308.911,A -85,B 0,C 180,E1 -14553.753,E2 -14553.753} C_VEL
LIN {X 0,Y 333.716,Z 308.912,A -85,B 0,C 180,E1 -14557.913,E2 -14557.913} C_VEL
LIN {X 0,Y 333.791,Z 308.905,A -85,B 0,C 180,E1 -14561.589,E2 -14561.589} C_VEL
LIN {X 0,Y 333.804,Z 308.904,A -85,B 0,C 180,E1 -14565.576,E2 -14565.576} C_VEL
LIN {X 0,Y 333.829,Z 308.899,A -85,B 0,C 180,E1 -14569.078,E2 -14569.078} C_VEL
LIN {X 0,Y 334.008,Z 308.876,A -85,B 0,C 180,E1 -14572.747,E2 -14572.747} C_VEL
LIN {X 0,Y 333.804,Z 308.903,A -85,B 0,C 180,E1 -14575.169,E2 -14575.169} C_VEL
LIN {X 0,Y 334.1,Z 308.869,A -85,B 0,C 180,E1 -14577.589,E2 -14577.589} C_VEL
LIN {X 0,Y 334.222,Z 308.851,A -85,B 0,C 180,E1 -14580,E2 -14580} C_VEL
LIN {X 0,Y 334.1,Z 308.865,A -85,B 0,C 180,E1 -14582.411,E2 -14582.411} C_VEL
LIN {X 0,Y 333.967,Z 308.882,A -85,B 0,C 180,E1 -14586.496,E2 -14586.496} C_VEL
LIN {X 0,Y 333.844,Z 308.898,A -85,B 0,C 180,E1 -14589.695,E2 -14589.695} C_VEL
LIN {X 0,Y 333.792,Z 308.903,A -85,B 0,C 180,E1 -14593.391,E2 -14593.391} C_VEL
LIN {X 0,Y 333.741,Z 308.909,A -85,B 0,C 180,E1 -14597.146,E2 -14597.146} C_VEL
LIN {X 0,Y 333.728,Z 308.91,A -85,B 0,C 180,E1 -14599.691,E2 -14599.691} C_VEL
LIN {X 0,Y 333.664,Z 308.919,A -85,B 0,C 180,E1 -14603.59,E2 -14603.59} C_VEL
LIN {X 0,Y 333.73,Z 308.915,A -85,B 0,C 180,E1 -14606.246,E2 -14606.246} C_VEL
LIN {X 0,Y 333.706,Z 308.914,A -85,B 0,C 180,E1 -14608.972,E2 -14608.972} C_VEL
LIN {X 0,Y 333.638,Z 308.927,A -85,B 0,C 180,E1 -14612.587,E2 -14612.587} C_VEL
LIN {X 0,Y 333.671,Z 308.919,A -85,B 0,C 180,E1 -14616.139,E2 -14616.139} C_VEL
LIN {X 0,Y 333.642,Z 308.923,A -85,B 0,C 180,E1 -14619.193,E2 -14619.193} C_VEL
LIN {X 0,Y 333.628,Z 308.925,A -85,B 0,C 180,E1 -14622.5,E2 -14622.5} C_VEL
LIN {X 0,Y 333.591,Z 308.926,A -85,B 0,C 180,E1 -14625.955,E2 -14625.955} C_VEL
LIN {X 0,Y 333.598,Z 308.93,A -85,B 0,C 180,E1 -14629.325,E2 -14629.325} C_VEL
LIN {X 0,Y 333.659,Z 308.925,A -85,B 0,C 180,E1 -14633.169,E2 -14633.169} C_VEL
LIN {X 0,Y 333.671,Z 308.923,A -85,B 0,C 180,E1 -14635.342,E2 -14635.342} C_VEL
LIN {X 0,Y 333.626,Z 308.923,A -85,B 0,C 180,E1 -14638.222,E2 -14638.222} C_VEL
LIN {X 0,Y 333.648,Z 308.923,A -85,B 0,C 180,E1 -14641.023,E2 -14641.023} C_VEL
LIN {X 0,Y 333.661,Z 308.921,A -85,B 0,C 180,E1 -14645.086,E2 -14645.086} C_VEL
LIN {X 0,Y 333.662,Z 308.92,A -85,B 0,C 180,E1 -14649.019,E2 -14649.019} C_VEL
LIN {X 0,Y 333.739,Z 308.915,A -85,B 0,C 180,E1 -14651.587,E2 -14651.587} C_VEL
LIN {X 0,Y 333.828,Z 309.021,A -85,B 0,C 180,E1 -14655.367,E2 -14655.367} C_VEL
LIN {X 0,Y 335.148,Z 315.537,A -85,B 0,C 180,E1 -14657.222,E2 -14657.222} C_VEL
LIN {X 0,Y 339.78,Z 330.155,A -85,B 0,C 180,E1 -14657.834,E2 -14657.834} C_VEL
LIN {X 0,Y 341.976,Z 343.835,A -85,B 0,C 180,E1 -14658.26,E2 -14658.26} C_VEL
LIN {X 0,Y 340.47,Z 423.067,A -85,B 0,C 180,E1 -14659.933,E2 -14659.933} C_VEL
LIN {X 0,Y 339.946,Z 436.183,A -85,B 0,C 180,E1 -14660.443,E2 -14660.443} C_VEL
LIN {X 0,Y 339.261,Z 449.338,A -85,B 0,C 180,E1 -14661.213,E2 -14661.213} C_VEL
LIN {X 0,Y 338.475,Z 460.424,A -85,B 0,C 180,E1 -14662.094,E2 -14662.094} C_VEL
LIN {X 0,Y 337.441,Z 469.409,A -85,B 0,C 180,E1 -14662.972,E2 -14662.972} C_VEL
LIN {X 0,Y 336.436,Z 480.229,A -85,B 0,C 180,E1 -14664.306,E2 -14664.306} C_VEL
LIN {X 0,Y 335.345,Z 489.961,A -85,B 0,C 180,E1 -14665.794,E2 -14665.794} C_VEL
LIN {X 0,Y 334.531,Z 497.927,A -85,B 0,C 180,E1 -14667.291,E2 -14667.291} C_VEL
LIN {X 0,Y 333.632,Z 505.767,A -85,B 0,C 180,E1 -14669.095,E2 -14669.095} C_VEL
LIN {X 0,Y 333.059,Z 511.078,A -85,B 0,C 180,E1 -14670.605,E2 -14670.605} C_VEL
LIN {X 0,Y 332.673,Z 516.265,A -85,B 0,C 180,E1 -14672.422,E2 -14672.422} C_VEL
LIN {X 0,Y 332.322,Z 520.311,A -85,B 0,C 180,E1 -14674.245,E2 -14674.245} C_VEL
LIN {X 0,Y 332.255,Z 523.478,A -85,B 0,C 180,E1 -14676.195,E2 -14676.195} C_VEL
LIN {X 0,Y 331.935,Z 525.813,A -85,B 0,C 180,E1 -14678.524,E2 -14678.524} C_VEL
LIN {X 0,Y 331.897,Z 526.724,A -85,B 0,C 180,E1 -14680.987,E2 -14680.987} C_VEL
LIN {X 0,Y 332.172,Z 526.077,A -85,B 0,C 180,E1 -14683.282,E2 -14683.282} C_VEL
LIN {X 0,Y 332.294,Z 524.985,A -85,B 0,C 180,E1 -14684.703,E2 -14684.703} C_VEL
LIN {X 0,Y 332.521,Z 523.593,A -85,B 0,C 180,E1 -14685.948,E2 -14685.948} C_VEL
LIN {X 0,Y 333.021,Z 520.715,A -85,B 0,C 180,E1 -14687.774,E2 -14687.774} C_VEL
LIN {X 0,Y 333.72,Z 516.586,A -85,B 0,C 180,E1 -14689.692,E2 -14689.692} C_VEL
LIN {X 0,Y 334.85,Z 510.285,A -85,B 0,C 180,E1 -14691.873,E2 -14691.873} C_VEL
LIN {X 0,Y 336.015,Z 503.365,A -85,B 0,C 180,E1 -14693.743,E2 -14693.743} C_VEL
LIN {X 0,Y 337.254,Z 496.253,A -85,B 0,C 180,E1 -14695.29,E2 -14695.29} C_VEL
LIN {X 0,Y 338.688,Z 487.556,A -85,B 0,C 180,E1 -14696.84,E2 -14696.84} C_VEL
LIN {X 0,Y 340.344,Z 476.851,A -85,B 0,C 180,E1 -14698.356,E2 -14698.356} C_VEL
LIN {X 0,Y 341.741,Z 466.094,A -85,B 0,C 180,E1 -14699.575,E2 -14699.575} C_VEL
LIN {X 0,Y 343.109,Z 453.851,A -85,B 0,C 180,E1 -14700.65,E2 -14700.65} C_VEL
LIN {X 0,Y 344.1,Z 441.383,A -85,B 0,C 180,E1 -14701.473,E2 -14701.473} C_VEL
LIN {X 0,Y 344.743,Z 428.238,A -85,B 0,C 180,E1 -14702.088,E2 -14702.088} C_VEL
LIN {X 0,Y 345.396,Z 413.749,A -85,B 0,C 180,E1 -14702.459,E2 -14702.459} C_VEL
LIN {X 0,Y 345.873,Z 393.016,A -85,B 0,C 180,E1 -14702.892,E2 -14702.892} C_VEL
LIN {X 0,Y 345.459,Z 387.21,A -85,B 0,C 180,E1 -14703.06,E2 -14703.06} C_VEL
LIN {X 0,Y 340.871,Z 368.545,A -85,B 0,C 180,E1 -14703.884,E2 -14703.884} C_VEL
LIN {X 0,Y 340.446,Z 362.739,A -85,B 0,C 180,E1 -14704.058,E2 -14704.058} C_VEL
LIN {X 0,Y 340.768,Z 346.277,A -85,B 0,C 180,E1 -14704.416,E2 -14704.416} C_VEL
LIN {X 0,Y 339.362,Z 341.125,A -85,B 0,C 180,E1 -14704.665,E2 -14704.665} C_VEL
LIN {X 0,Y 331.366,Z 322.862,A -85,B 0,C 180,E1 -14705.865,E2 -14705.865} C_VEL
LIN {X 0,Y 328.226,Z 316.231,A -85,B 0,C 180,E1 -14706.378,E2 -14706.378} C_VEL
LIN {X 0,Y 326.643,Z 309.793,A -85,B 0,C 180,E1 -14708.522,E2 -14708.522} C_VEL
LIN {X 0,Y 326.575,Z 309.803,A -85,B 0,C 180,E1 -14711.846,E2 -14711.846} C_VEL
LIN {X 0,Y 326.527,Z 309.812,A -85,B 0,C 180,E1 -14715.257,E2 -14715.257} C_VEL
LIN {X 0,Y 326.577,Z 309.804,A -85,B 0,C 180,E1 -14718.869,E2 -14718.869} C_VEL
LIN {X 0,Y 326.627,Z 309.797,A -85,B 0,C 180,E1 -14722.762,E2 -14722.762} C_VEL
LIN {X 0,Y 326.606,Z 309.794,A -85,B 0,C 180,E1 -14725.981,E2 -14725.981} C_VEL
LIN {X 0,Y 326.66,Z 309.786,A -85,B 0,C 180,E1 -14730.341,E2 -14730.341} C_VEL
LIN {X 0,Y 326.69,Z 309.784,A -85,B 0,C 180,E1 -14734.516,E2 -14734.516} C_VEL
LIN {X 0,Y 326.62,Z 309.795,A -85,B 0,C 180,E1 -14738.544,E2 -14738.544} C_VEL
LIN {X 0,Y 326.744,Z 309.776,A -85,B 0,C 180,E1 -14741.178,E2 -14741.178} C_VEL
LIN {X 0,Y 326.763,Z 309.776,A -85,B 0,C 180,E1 -14745.433,E2 -14745.433} C_VEL
LIN {X 0,Y 326.77,Z 309.774,A -85,B 0,C 180,E1 -14748.839,E2 -14748.839} C_VEL
LIN {X 0,Y 326.979,Z 309.749,A -85,B 0,C 180,E1 -14752.591,E2 -14752.591} C_VEL
LIN {X 0,Y 326.777,Z 309.776,A -85,B 0,C 180,E1 -14755.065,E2 -14755.065} C_VEL
LIN {X 0,Y 327.046,Z 309.74,A -85,B 0,C 180,E1 -14757.537,E2 -14757.537} C_VEL
LIN {X 0,Y 327.179,Z 309.729,A -85,B 0,C 180,E1 -14760,E2 -14760} C_VEL
LIN {X 0,Y 327.046,Z 309.737,A -85,B 0,C 180,E1 -14762.464,E2 -14762.464} C_VEL
LIN {X 0,Y 326.995,Z 309.746,A -85,B 0,C 180,E1 -14766.169,E2 -14766.169} C_VEL
LIN {X 0,Y 326.915,Z 309.761,A -85,B 0,C 180,E1 -14768.655,E2 -14768.655} C_VEL
LIN {X 0,Y 326.735,Z 309.777,A -85,B 0,C 180,E1 -14772.422,E2 -14772.422} C_VEL
LIN {X 0,Y 326.755,Z 309.776,A -85,B 0,C 180,E1 -14774.958,E2 -14774.958} C_VEL
LIN {X 0,Y 326.733,Z 309.783,A -85,B 0,C 180,E1 -14778.838,E2 -14778.838} C_VEL
LIN {X 0,Y 326.604,Z 309.803,A -85,B 0,C 180,E1 -14782.789,E2 -14782.789} C_VEL
LIN {X 0,Y 326.691,Z 309.788,A -85,B 0,C 180,E1 -14785.484,E2 -14785.484} C_VEL
LIN {X 0,Y 326.661,Z 309.793,A -85,B 0,C 180,E1 -14789.659,E2 -14789.659} C_VEL
LIN {X 0,Y 326.608,Z 309.799,A -85,B 0,C 180,E1 -14794.02,E2 -14794.02} C_VEL
LIN {X 0,Y 326.629,Z 309.799,A -85,B 0,C 180,E1 -14797.239,E2 -14797.239} C_VEL
LIN {X 0,Y 326.579,Z 309.784,A -85,B 0,C 180,E1 -14801.131,E2 -14801.131} C_VEL
LIN {X 0,Y 326.529,Z 309.807,A -85,B 0,C 180,E1 -14804.743,E2 -14804.743} C_VEL
LIN {X 0,Y 326.578,Z 309.805,A -85,B 0,C 180,E1 -14808.154,E2 -14808.154} C_VEL
LIN {X 0,Y 326.625,Z 309.801,A -85,B 0,C 180,E1 -14811.392,E2 -14811.392} C_VEL
LIN {X 0,Y 326.64,Z 309.793,A -85,B 0,C 180,E1 -14815.237,E2 -14815.237} C_VEL
LIN {X 0,Y 326.638,Z 309.924,A -85,B 0,C 180,E1 -14815.891,E2 -14815.891} C_VEL
LIN {X 0,Y 329.578,Z 321.739,A -85,B 0,C 180,E1 -14819.573,E2 -14819.573} C_VEL
LIN {X 0,Y 331.941,Z 332.735,A -85,B 0,C 180,E1 -14822.779,E2 -14822.779} C_VEL
LIN {X 0,Y 332.358,Z 335.839,A -85,B 0,C 180,E1 -14823.636,E2 -14823.636} C_VEL
LIN {X 0,Y 332.141,Z 337.673,A -85,B 0,C 180,E1 -14824.099,E2 -14824.099} C_VEL
LIN {X 0,Y 337.575,Z 363.518,A -85,B 0,C 180,E1 -14825.237,E2 -14825.237} C_VEL
LIN {X 0,Y 340.084,Z 379.469,A -85,B 0,C 180,E1 -14825.836,E2 -14825.836} C_VEL
LIN {X 0,Y 338.397,Z 446.39,A -85,B 0,C 180,E1 -14827.284,E2 -14827.284} C_VEL
LIN {X 0,Y 337.504,Z 459.587,A -85,B 0,C 180,E1 -14827.785,E2 -14827.785} C_VEL
LIN {X 0,Y 336.23,Z 472.823,A -85,B 0,C 180,E1 -14828.543,E2 -14828.543} C_VEL
LIN {X 0,Y 334.949,Z 483.953,A -85,B 0,C 180,E1 -14829.423,E2 -14829.423} C_VEL
LIN {X 0,Y 333.196,Z 495.528,A -85,B 0,C 180,E1 -14830.597,E2 -14830.597} C_VEL
LIN {X 0,Y 331.556,Z 505.954,A -85,B 0,C 180,E1 -14831.94,E2 -14831.94} C_VEL
LIN {X 0,Y 329.885,Z 515.545,A -85,B 0,C 180,E1 -14833.477,E2 -14833.477} C_VEL
LIN {X 0,Y 328.628,Z 523.788,A -85,B 0,C 180,E1 -14835.129,E2 -14835.129} C_VEL
LIN {X 0,Y 327.264,Z 531.256,A -85,B 0,C 180,E1 -14836.968,E2 -14836.968} C_VEL
LIN {X 0,Y 326.29,Z 537.279,A -85,B 0,C 180,E1 -14838.822,E2 -14838.822} C_VEL
LIN {X 0,Y 325.593,Z 542.064,A -85,B 0,C 180,E1 -14840.683,E2 -14840.683} C_VEL
LIN {X 0,Y 325.157,Z 545.75,A -85,B 0,C 180,E1 -14842.548,E2 -14842.548} C_VEL
LIN {X 0,Y 324.926,Z 548.24,A -85,B 0,C 180,E1 -14844.248,E2 -14844.248} C_VEL
LIN {X 0,Y 324.902,Z 550.193,A -85,B 0,C 180,E1 -14846.279,E2 -14846.279} C_VEL
LIN {X 0,Y 324.872,Z 551.135,A -85,B 0,C 180,E1 -14848.76,E2 -14848.76} C_VEL
LIN {X 0,Y 324.948,Z 551.008,A -85,B 0,C 180,E1 -14850,E2 -14850} C_VEL
LIN {X 0,Y 324.903,Z 550.45,A -85,B 0,C 180,E1 -14851.239,E2 -14851.239} C_VEL
LIN {X 0,Y 324.945,Z 548.153,A -85,B 0,C 180,E1 -14853.72,E2 -14853.72} C_VEL
LIN {X 0,Y 324.992,Z 544.773,A -85,B 0,C 180,E1 -14855.867,E2 -14855.867} C_VEL
LIN {X 0,Y 325.226,Z 539.8,A -85,B 0,C 180,E1 -14858.074,E2 -14858.074} C_VEL
LIN {X 0,Y 325.7,Z 533.288,A -85,B 0,C 180,E1 -14860.254,E2 -14860.254} C_VEL
LIN {X 0,Y 326.407,Z 526.136,A -85,B 0,C 180,E1 -14862.118,E2 -14862.118} C_VEL
LIN {X 0,Y 327.373,Z 517.199,A -85,B 0,C 180,E1 -14863.975,E2 -14863.975} C_VEL
LIN {X 0,Y 328.361,Z 508.66,A -85,B 0,C 180,E1 -14865.416,E2 -14865.416} C_VEL
LIN {X 0,Y 329.397,Z 497.856,A -85,B 0,C 180,E1 -14866.899,E2 -14866.899} C_VEL
LIN {X 0,Y 330.599,Z 486.556,A -85,B 0,C 180,E1 -14868.113,E2 -14868.113} C_VEL
LIN {X 0,Y 331.747,Z 473.845,A -85,B 0,C 180,E1 -14869.169,E2 -14869.169} C_VEL
LIN {X 0,Y 332.674,Z 461.437,A -85,B 0,C 180,E1 -14869.916,E2 -14869.916} C_VEL
LIN {X 0,Y 333.441,Z 447.623,A -85,B 0,C 180,E1 -14870.471,E2 -14870.471} C_VEL
LIN {X 0,Y 334.641,Z 376.801,A -85,B 0,C 180,E1 -14872.017,E2 -14872.017} C_VEL
LIN {X 0,Y 329.35,Z 338.251,A -85,B 0,C 180,E1 -14873.215,E2 -14873.215} C_VEL
LIN {X 0,Y 330.303,Z 328.793,A -85,B 0,C 180,E1 -14875.522,E2 -14875.522} C_VEL
LIN {X 0,Y 328.938,Z 320.572,A -85,B 0,C 180,E1 -14877.69,E2 -14877.69} C_VEL
LIN {X 0,Y 326.634,Z 309.803,A -85,B 0,C 180,E1 -14880.663,E2 -14880.663} C_VEL
LIN {X 0,Y 326.606,Z 309.803,A -85,B 0,C 180,E1 -14884.019,E2 -14884.019} C_VEL
LIN {X 0,Y 326.626,Z 309.796,A -85,B 0,C 180,E1 -14887.238,E2 -14887.238} C_VEL
LIN {X 0,Y 326.576,Z 309.802,A -85,B 0,C 180,E1 -14891.13,E2 -14891.13} C_VEL
LIN {X 0,Y 326.525,Z 309.812,A -85,B 0,C 180,E1 -14894.742,E2 -14894.742} C_VEL
LIN {X 0,Y 326.574,Z 309.804,A -85,B 0,C 180,E1 -14898.153,E2 -14898.153} C_VEL
LIN {X 0,Y 326.595,Z 309.8,A -85,B 0,C 180,E1 -14901.387,E2 -14901.387} C_VEL
LIN {X 0,Y 326.617,Z 309.802,A -85,B 0,C 180,E1 -14904.85,E2 -14904.85} C_VEL
LIN {X 0,Y 326.605,Z 309.799,A -85,B 0,C 180,E1 -14907.455,E2 -14907.455} C_VEL
LIN {X 0,Y 326.644,Z 309.795,A -85,B 0,C 180,E1 -14910.339,E2 -14910.339} C_VEL
LIN {X 0,Y 326.687,Z 309.79,A -85,B 0,C 180,E1 -14914.516,E2 -14914.516} C_VEL
LIN {X 0,Y 326.643,Z 309.794,A -85,B 0,C 180,E1 -14918.545,E2 -14918.545} C_VEL
LIN {X 0,Y 326.741,Z 309.787,A -85,B 0,C 180,E1 -14921.177,E2 -14921.177} C_VEL
LIN {X 0,Y 326.759,Z 309.783,A -85,B 0,C 180,E1 -14925.433,E2 -14925.433} C_VEL
LIN {X 0,Y 326.765,Z 309.776,A -85,B 0,C 180,E1 -14928.839,E2 -14928.839} C_VEL
LIN {X 0,Y 326.962,Z 309.753,A -85,B 0,C 180,E1 -14932.59,E2 -14932.59} C_VEL
LIN {X 0,Y 326.771,Z 309.779,A -85,B 0,C 180,E1 -14935.064,E2 -14935.064} C_VEL
LIN {X 0,Y 327.041,Z 309.748,A -85,B 0,C 180,E1 -14937.536,E2 -14937.536} C_VEL
LIN {X 0,Y 327.174,Z 309.729,A -85,B 0,C 180,E1 -14940,E2 -14940} C_VEL
LIN {X 0,Y 327.041,Z 309.744,A -85,B 0,C 180,E1 -14942.463,E2 -14942.463} C_VEL
LIN {X 0,Y 326.927,Z 309.758,A -85,B 0,C 180,E1 -14946.485,E2 -14946.485} C_VEL
LIN {X 0,Y 326.8,Z 309.776,A -85,B 0,C 180,E1 -14949.906,E2 -14949.906} C_VEL
LIN {X 0,Y 326.754,Z 309.781,A -85,B 0,C 180,E1 -14953.685,E2 -14953.685} C_VEL
LIN {X 0,Y 326.694,Z 309.787,A -85,B 0,C 180,E1 -14957.528,E2 -14957.528} C_VEL
LIN {X 0,Y 326.653,Z 309.795,A -85,B 0,C 180,E1 -14960.135,E2 -14960.135} C_VEL
LIN {X 0,Y 326.643,Z 309.796,A -85,B 0,C 180,E1 -14964.129,E2 -14964.129} C_VEL
LIN {X 0,Y 326.68,Z 309.79,A -85,B 0,C 180,E1 -14966.858,E2 -14966.858} C_VEL
LIN {X 0,Y 326.634,Z 309.798,A -85,B 0,C 180,E1 -14970.611,E2 -14970.611} C_VEL
LIN {X 0,Y 326.602,Z 309.799,A -85,B 0,C 180,E1 -14974.02,E2 -14974.02} C_VEL
LIN {X 0,Y 326.623,Z 309.796,A -85,B 0,C 180,E1 -14977.239,E2 -14977.239} C_VEL
LIN {X 0,Y 326.573,Z 309.805,A -85,B 0,C 180,E1 -14981.132,E2 -14981.132} C_VEL
LIN {X 0,Y 326.523,Z 309.812,A -85,B 0,C 180,E1 -14984.743,E2 -14984.743} C_VEL
LIN {X 0,Y 326.558,Z 309.804,A -85,B 0,C 180,E1 -14988.152,E2 -14988.152} C_VEL
LIN {X 0,Y 326.578,Z 309.804,A -85,B 0,C 180,E1 -14991.386,E2 -14991.386} C_VEL
LIN {X 0,Y 326.616,Z 309.799,A -85,B 0,C 180,E1 -14994.852,E2 -14994.852} C_VEL
LIN {X 0,Y 326.605,Z 309.803,A -85,B 0,C 180,E1 -14997.456,E2 -14997.456} C_VEL
LIN {X 0,Y 326.586,Z 309.799,A -85,B 0,C 180,E1 -15000.334,E2 -15000.334} C_VEL
LIN {X 0,Y 326.594,Z 309.802,A -85,B 0,C 180,E1 -15003.135,E2 -15003.135} C_VEL
LIN {X 0,Y 326.59,Z 309.803,A -85,B 0,C 180,E1 -15007.211,E2 -15007.211} C_VEL
LIN {X 0,Y 326.705,Z 309.788,A -85,B 0,C 180,E1 -15011.176,E2 -15011.176} C_VEL
LIN {X 0,Y 326.784,Z 309.834,A -85,B 0,C 180,E1 -15015.045,E2 -15015.045} C_VEL
LIN {X 0,Y 328.017,Z 315.819,A -85,B 0,C 180,E1 -15016.79,E2 -15016.79} C_VEL
LIN {X 0,Y 333.26,Z 332.18,A -85,B 0,C 180,E1 -15017.492,E2 -15017.492} C_VEL
LIN {X 0,Y 335.268,Z 344.12,A -85,B 0,C 180,E1 -15017.879,E2 -15017.879} C_VEL
LIN {X 0,Y 333.706,Z 422.996,A -85,B 0,C 180,E1 -15019.573,E2 -15019.573} C_VEL
LIN {X 0,Y 333.165,Z 436.225,A -85,B 0,C 180,E1 -15020.093,E2 -15020.093} C_VEL
LIN {X 0,Y 332.457,Z 449.439,A -85,B 0,C 180,E1 -15020.878,E2 -15020.878} C_VEL
LIN {X 0,Y 331.642,Z 460.57,A -85,B 0,C 180,E1 -15021.777,E2 -15021.777} C_VEL
LIN {X 0,Y 330.591,Z 469.566,A -85,B 0,C 180,E1 -15022.672,E2 -15022.672} C_VEL
LIN {X 0,Y 329.667,Z 479.347,A -85,B 0,C 180,E1 -15023.882,E2 -15023.882} C_VEL
LIN {X 0,Y 328.491,Z 489.279,A -85,B 0,C 180,E1 -15025.399,E2 -15025.399} C_VEL
LIN {X 0,Y 327.475,Z 498.881,A -85,B 0,C 180,E1 -15027.233,E2 -15027.233} C_VEL
LIN {X 0,Y 326.547,Z 506.555,A -85,B 0,C 180,E1 -15029.076,E2 -15029.076} C_VEL
LIN {X 0,Y 325.851,Z 513.608,A -85,B 0,C 180,E1 -15031.236,E2 -15031.236} C_VEL
LIN {X 0,Y 325.377,Z 518.317,A -85,B 0,C 180,E1 -15033.096,E2 -15033.096} C_VEL
LIN {X 0,Y 325.215,Z 521.912,A -85,B 0,C 180,E1 -15034.959,E2 -15034.959} C_VEL
LIN {X 0,Y 325.154,Z 523.771,A -85,B 0,C 180,E1 -15036.205,E2 -15036.205} C_VEL
LIN {X 0,Y 324.966,Z 525.173,A -85,B 0,C 180,E1 -15037.456,E2 -15037.456} C_VEL
LIN {X 0,Y 324.77,Z 526.787,A -85,B 0,C 180,E1 -15039.97,E2 -15039.97} C_VEL
LIN {X 0,Y 324.823,Z 526.992,A -85,B 0,C 180,E1 -15041.229,E2 -15041.229} C_VEL
LIN {X 0,Y 325.076,Z 526.376,A -85,B 0,C 180,E1 -15043.375,E2 -15043.375} C_VEL
LIN {X 0,Y 325.263,Z 525.12,A -85,B 0,C 180,E1 -15045.028,E2 -15045.028} C_VEL
LIN {X 0,Y 325.514,Z 523.654,A -85,B 0,C 180,E1 -15046.301,E2 -15046.301} C_VEL
LIN {X 0,Y 326.211,Z 519.914,A -85,B 0,C 180,E1 -15048.568,E2 -15048.568} C_VEL
LIN {X 0,Y 327.157,Z 514.837,A -85,B 0,C 180,E1 -15050.76,E2 -15050.76} C_VEL
LIN {X 0,Y 328.243,Z 509.029,A -85,B 0,C 180,E1 -15052.669,E2 -15052.669} C_VEL
LIN {X 0,Y 329.547,Z 501.671,A -85,B 0,C 180,E1 -15054.574,E2 -15054.574} C_VEL
LIN {X 0,Y 331.245,Z 492.478,A -85,B 0,C 180,E1 -15056.459,E2 -15056.459} C_VEL
LIN {X 0,Y 332.854,Z 482.88,A -85,B 0,C 180,E1 -15058.021,E2 -15058.021} C_VEL
LIN {X 0,Y 334.473,Z 472.127,A -85,B 0,C 180,E1 -15059.417,E2 -15059.417} C_VEL
LIN {X 0,Y 335.998,Z 460.305,A -85,B 0,C 180,E1 -15060.627,E2 -15060.627} C_VEL
LIN {X 0,Y 337.217,Z 448.083,A -85,B 0,C 180,E1 -15061.576,E2 -15061.576} C_VEL
LIN {X 0,Y 338.122,Z 435.146,A -85,B 0,C 180,E1 -15062.315,E2 -15062.315} C_VEL
LIN {X 0,Y 338.582,Z 424.512,A -85,B 0,C 180,E1 -15062.732,E2 -15062.732} C_VEL
LIN {X 0,Y 339.501,Z 394.669,A -85,B 0,C 180,E1 -15063.392,E2 -15063.392} C_VEL
LIN {X 0,Y 340.446,Z 362.739,A -85,B 0,C 180,E1 -15064.058,E2 -15064.058} C_VEL
LIN {X 0,Y 340.075,Z 358.88,A -85,B 0,C 180,E1 -15064.182,E2 -15064.182} C_VEL
LIN {X 0,Y 337.973,Z 352.902,A -85,B 0,C 180,E1 -15064.513,E2 -15064.513} C_VEL
LIN {X 0,Y 333.393,Z 343.714,A -85,B 0,C 180,E1 -15065.16,E2 -15065.16} C_VEL
LIN {X 0,Y 325.981,Z 326.744,A -85,B 0,C 180,E1 -15066.309,E2 -15066.309} C_VEL
LIN {X 0,Y 321.061,Z 316.619,A -85,B 0,C 180,E1 -15067.098,E2 -15067.098} C_VEL
LIN {X 0,Y 319.575,Z 310.681,A -85,B 0,C 180,E1 -15069.116,E2 -15069.116} C_VEL
LIN {X 0,Y 319.553,Z 310.682,A -85,B 0,C 180,E1 -15072.984,E2 -15072.984} C_VEL
LIN {X 0,Y 319.553,Z 310.68,A -85,B 0,C 180,E1 -15077.017,E2 -15077.017} C_VEL
LIN {X 0,Y 319.546,Z 310.678,A -85,B 0,C 180,E1 -15080.371,E2 -15080.371} C_VEL
LIN {X 0,Y 319.579,Z 310.673,A -85,B 0,C 180,E1 -15084.457,E2 -15084.457} C_VEL
LIN {X 0,Y 319.532,Z 310.674,A -85,B 0,C 180,E1 -15088.138,E2 -15088.138} C_VEL
LIN {X 0,Y 319.615,Z 310.663,A -85,B 0,C 180,E1 -15091.589,E2 -15091.589} C_VEL
LIN {X 0,Y 319.603,Z 310.667,A -85,B 0,C 180,E1 -15095.304,E2 -15095.304} C_VEL
LIN {X 0,Y 319.602,Z 310.669,A -85,B 0,C 180,E1 -15099.401,E2 -15099.401} C_VEL
LIN {X 0,Y 319.658,Z 310.666,A -85,B 0,C 180,E1 -15102.073,E2 -15102.073} C_VEL
LIN {X 0,Y 319.732,Z 310.658,A -85,B 0,C 180,E1 -15106.008,E2 -15106.008} C_VEL
LIN {X 0,Y 319.758,Z 310.65,A -85,B 0,C 180,E1 -15109.873,E2 -15109.873} C_VEL
LIN {X 0,Y 319.933,Z 310.627,A -85,B 0,C 180,E1 -15112.426,E2 -15112.426} C_VEL
LIN {X 0,Y 319.746,Z 310.652,A -85,B 0,C 180,E1 -15114.956,E2 -15114.956} C_VEL
LIN {X 0,Y 319.99,Z 310.619,A -85,B 0,C 180,E1 -15117.483,E2 -15117.483} C_VEL
LIN {X 0,Y 320.132,Z 310.607,A -85,B 0,C 180,E1 -15120,E2 -15120} C_VEL
LIN {X 0,Y 319.989,Z 310.615,A -85,B 0,C 180,E1 -15122.518,E2 -15122.518} C_VEL
LIN {X 0,Y 319.951,Z 310.622,A -85,B 0,C 180,E1 -15126.306,E2 -15126.306} C_VEL
LIN {X 0,Y 319.843,Z 310.641,A -85,B 0,C 180,E1 -15128.848,E2 -15128.848} C_VEL
LIN {X 0,Y 319.682,Z 310.658,A -85,B 0,C 180,E1 -15132.7,E2 -15132.7} C_VEL
LIN {X 0,Y 319.7,Z 310.653,A -85,B 0,C 180,E1 -15135.296,E2 -15135.296} C_VEL
LIN {X 0,Y 319.674,Z 310.659,A -85,B 0,C 180,E1 -15139.255,E2 -15139.255} C_VEL
LIN {X 0,Y 319.561,Z 310.675,A -85,B 0,C 180,E1 -15143.32,E2 -15143.32} C_VEL
LIN {X 0,Y 319.635,Z 310.667,A -85,B 0,C 180,E1 -15146.088,E2 -15146.088} C_VEL
LIN {X 0,Y 319.59,Z 310.67,A -85,B 0,C 180,E1 -15148.934,E2 -15148.934} C_VEL
LIN {X 0,Y 319.533,Z 310.677,A -85,B 0,C 180,E1 -15151.862,E2 -15151.862} C_VEL
LIN {X 0,Y 319.581,Z 310.67,A -85,B 0,C 180,E1 -15155.543,E2 -15155.543} C_VEL
LIN {X 0,Y 319.558,Z 310.676,A -85,B 0,C 180,E1 -15158.01,E2 -15158.01} C_VEL
LIN {X 0,Y 319.527,Z 310.667,A -85,B 0,C 180,E1 -15161.597,E2 -15161.597} C_VEL
LIN {X 0,Y 319.49,Z 310.687,A -85,B 0,C 180,E1 -15165.257,E2 -15165.257} C_VEL
LIN {X 0,Y 319.53,Z 310.682,A -85,B 0,C 180,E1 -15168.712,E2 -15168.712} C_VEL
LIN {X 0,Y 319.563,Z 310.672,A -85,B 0,C 180,E1 -15172.348,E2 -15172.348} C_VEL
LIN {X 0,Y 319.611,Z 310.806,A -85,B 0,C 180,E1 -15175.269,E2 -15175.269} C_VEL
LIN {X 0,Y 322.681,Z 323.104,A -85,B 0,C 180,E1 -15179.214,E2 -15179.214} C_VEL
LIN {X 0,Y 324.993,Z 333.927,A -85,B 0,C 180,E1 -15182.453,E2 -15182.453} C_VEL
LIN {X 0,Y 325.544,Z 337.555,A -85,B 0,C 180,E1 -15183.452,E2 -15183.452} C_VEL
LIN {X 0,Y 330.45,Z 360.148,A -85,B 0,C 180,E1 -15184.493,E2 -15184.493} C_VEL
LIN {X 0,Y 333.788,Z 380.186,A -85,B 0,C 180,E1 -15185.291,E2 -15185.291} C_VEL
LIN {X 0,Y 332.043,Z 446.108,A -85,B 0,C 180,E1 -15186.741,E2 -15186.741} C_VEL
LIN {X 0,Y 331.129,Z 459.302,A -85,B 0,C 180,E1 -15187.252,E2 -15187.252} C_VEL
LIN {X 0,Y 329.922,Z 471.419,A -85,B 0,C 180,E1 -15187.948,E2 -15187.948} C_VEL
LIN {X 0,Y 328.558,Z 482.845,A -85,B 0,C 180,E1 -15188.84,E2 -15188.84} C_VEL
LIN {X 0,Y 326.755,Z 494.6,A -85,B 0,C 180,E1 -15190.035,E2 -15190.035} C_VEL
LIN {X 0,Y 324.997,Z 505.139,A -85,B 0,C 180,E1 -15191.399,E2 -15191.399} C_VEL
LIN {X 0,Y 323.205,Z 515.009,A -85,B 0,C 180,E1 -15192.994,E2 -15192.994} C_VEL
LIN {X 0,Y 321.746,Z 523.849,A -85,B 0,C 180,E1 -15194.804,E2 -15194.804} C_VEL
LIN {X 0,Y 320.351,Z 531.26,A -85,B 0,C 180,E1 -15196.682,E2 -15196.682} C_VEL
LIN {X 0,Y 319.278,Z 537.231,A -85,B 0,C 180,E1 -15198.573,E2 -15198.573} C_VEL
LIN {X 0,Y 318.575,Z 541.97,A -85,B 0,C 180,E1 -15200.476,E2 -15200.476} C_VEL
LIN {X 0,Y 318.085,Z 545.612,A -85,B 0,C 180,E1 -15202.382,E2 -15202.382} C_VEL
LIN {X 0,Y 317.845,Z 548.248,A -85,B 0,C 180,E1 -15204.28,E2 -15204.28} C_VEL
LIN {X 0,Y 317.809,Z 549.975,A -85,B 0,C 180,E1 -15206.196,E2 -15206.196} C_VEL
LIN {X 0,Y 317.778,Z 550.62,A -85,B 0,C 180,E1 -15207.464,E2 -15207.464} C_VEL
LIN {X 0,Y 317.781,Z 550.879,A -85,B 0,C 180,E1 -15208.732,E2 -15208.732} C_VEL
LIN {X 0,Y 317.853,Z 550.714,A -85,B 0,C 180,E1 -15210,E2 -15210} C_VEL
LIN {X 0,Y 317.811,Z 550.137,A -85,B 0,C 180,E1 -15211.267,E2 -15211.267} C_VEL
LIN {X 0,Y 317.801,Z 549.168,A -85,B 0,C 180,E1 -15212.534,E2 -15212.534} C_VEL
LIN {X 0,Y 317.85,Z 547.801,A -85,B 0,C 180,E1 -15213.803,E2 -15213.803} C_VEL
LIN {X 0,Y 317.889,Z 544.735,A -85,B 0,C 180,E1 -15215.799,E2 -15215.799} C_VEL
LIN {X 0,Y 318.061,Z 540.927,A -85,B 0,C 180,E1 -15217.618,E2 -15217.618} C_VEL
LIN {X 0,Y 318.498,Z 534.817,A -85,B 0,C 180,E1 -15219.846,E2 -15219.846} C_VEL
LIN {X 0,Y 319.129,Z 528.11,A -85,B 0,C 180,E1 -15221.753,E2 -15221.753} C_VEL
LIN {X 0,Y 320.111,Z 519.781,A -85,B 0,C 180,E1 -15223.651,E2 -15223.651} C_VEL
LIN {X 0,Y 321.249,Z 510.045,A -85,B 0,C 180,E1 -15225.415,E2 -15225.415} C_VEL
LIN {X 0,Y 322.255,Z 499.43,A -85,B 0,C 180,E1 -15226.959,E2 -15226.959} C_VEL
LIN {X 0,Y 323.439,Z 488.679,A -85,B 0,C 180,E1 -15228.2,E2 -15228.2} C_VEL
LIN {X 0,Y 324.681,Z 476.623,A -85,B 0,C 180,E1 -15229.274,E2 -15229.274} C_VEL
LIN {X 0,Y 325.66,Z 464.03,A -85,B 0,C 180,E1 -15230.117,E2 -15230.117} C_VEL
LIN {X 0,Y 326.523,Z 450.856,A -85,B 0,C 180,E1 -15230.719,E2 -15230.719} C_VEL
LIN {X 0,Y 326.868,Z 434.754,A -85,B 0,C 180,E1 -15231.15,E2 -15231.15} C_VEL
LIN {X 0,Y 327.971,Z 378.258,A -85,B 0,C 180,E1 -15232.37,E2 -15232.37} C_VEL
LIN {X 0,Y 322.492,Z 337.958,A -85,B 0,C 180,E1 -15233.658,E2 -15233.658} C_VEL
LIN {X 0,Y 323.3,Z 329.506,A -85,B 0,C 180,E1 -15235.77,E2 -15235.77} C_VEL
LIN {X 0,Y 321.581,Z 319.896,A -85,B 0,C 180,E1 -15238.38,E2 -15238.38} C_VEL
LIN {X 0,Y 319.574,Z 310.681,A -85,B 0,C 180,E1 -15241.016,E2 -15241.016} C_VEL
LIN {X 0,Y 319.559,Z 310.677,A -85,B 0,C 180,E1 -15244.876,E2 -15244.876} C_VEL
LIN {X 0,Y 319.572,Z 310.678,A -85,B 0,C 180,E1 -15248.007,E2 -15248.007} C_VEL
LIN {X 0,Y 319.524,Z 310.681,A -85,B 0,C 180,E1 -15251.596,E2 -15251.596} C_VEL
LIN {X 0,Y 319.486,Z 310.686,A -85,B 0,C 180,E1 -15255.256,E2 -15255.256} C_VEL
LIN {X 0,Y 319.527,Z 310.685,A -85,B 0,C 180,E1 -15258.711,E2 -15258.711} C_VEL
LIN {X 0,Y 319.551,Z 310.68,A -85,B 0,C 180,E1 -15262.349,E2 -15262.349} C_VEL
LIN {X 0,Y 319.557,Z 310.679,A -85,B 0,C 180,E1 -15265.123,E2 -15265.123} C_VEL
LIN {X 0,Y 319.563,Z 310.68,A -85,B 0,C 180,E1 -15269.058,E2 -15269.058} C_VEL
LIN {X 0,Y 319.602,Z 310.672,A -85,B 0,C 180,E1 -15272.497,E2 -15272.497} C_VEL
LIN {X 0,Y 319.602,Z 310.674,A -85,B 0,C 180,E1 -15275.303,E2 -15275.303} C_VEL
LIN {X 0,Y 319.593,Z 310.671,A -85,B 0,C 180,E1 -15278.047,E2 -15278.047} C_VEL
LIN {X 0,Y 319.686,Z 310.664,A -85,B 0,C 180,E1 -15280.961,E2 -15280.961} C_VEL
LIN {X 0,Y 319.727,Z 310.661,A -85,B 0,C 180,E1 -15285.275,E2 -15285.275} C_VEL
LIN {X 0,Y 319.753,Z 310.652,A -85,B 0,C 180,E1 -15289.872,E2 -15289.872} C_VEL
LIN {X 0,Y 319.921,Z 310.63,A -85,B 0,C 180,E1 -15292.426,E2 -15292.426} C_VEL
LIN {X 0,Y 319.74,Z 310.654,A -85,B 0,C 180,E1 -15294.956,E2 -15294.956} C_VEL
LIN {X 0,Y 319.984,Z 310.626,A -85,B 0,C 180,E1 -15297.482,E2 -15297.482} C_VEL
LIN {X 0,Y 320.126,Z 310.606,A -85,B 0,C 180,E1 -15300,E2 -15300} C_VEL
LIN {X 0,Y 319.985,Z 310.623,A -85,B 0,C 180,E1 -15302.517,E2 -15302.517} C_VEL
LIN {X 0,Y 319.893,Z 310.634,A -85,B 0,C 180,E1 -15306.469,E2 -15306.469} C_VEL
LIN {X 0,Y 319.747,Z 310.654,A -85,B 0,C 180,E1 -15310.127,E2 -15310.127} C_VEL
LIN {X 0,Y 319.726,Z 310.656,A -85,B 0,C 180,E1 -15314.724,E2 -15314.724} C_VEL
LIN {X 0,Y 319.684,Z 310.658,A -85,B 0,C 180,E1 -15319.038,E2 -15319.038} C_VEL
LIN {X 0,Y 319.555,Z 310.676,A -85,B 0,C 180,E1 -15323.32,E2 -15323.32} C_VEL
LIN {X 0,Y 319.63,Z 310.67,A -85,B 0,C 180,E1 -15326.088,E2 -15326.088} C_VEL
LIN {X 0,Y 319.584,Z 310.671,A -85,B 0,C 180,E1 -15328.934,E2 -15328.934} C_VEL
LIN {X 0,Y 319.527,Z 310.678,A -85,B 0,C 180,E1 -15331.862,E2 -15331.862} C_VEL
LIN {X 0,Y 319.575,Z 310.674,A -85,B 0,C 180,E1 -15335.543,E2 -15335.543} C_VEL
LIN {X 0,Y 319.554,Z 310.674,A -85,B 0,C 180,E1 -15339.669,E2 -15339.669} C_VEL
LIN {X 0,Y 319.517,Z 310.682,A -85,B 0,C 180,E1 -15343.461,E2 -15343.461} C_VEL
LIN {X 0,Y 319.548,Z 310.681,A -85,B 0,C 180,E1 -15347.017,E2 -15347.017} C_VEL
LIN {X 0,Y 319.541,Z 310.678,A -85,B 0,C 180,E1 -15350.371,E2 -15350.371} C_VEL
LIN {X 0,Y 319.576,Z 310.674,A -85,B 0,C 180,E1 -15354.458,E2 -15354.458} C_VEL
LIN {X 0,Y 319.521,Z 310.681,A -85,B 0,C 180,E1 -15358.138,E2 -15358.138} C_VEL
LIN {X 0,Y 319.565,Z 310.678,A -85,B 0,C 180,E1 -15361.605,E2 -15361.605} C_VEL
LIN {X 0,Y 319.539,Z 310.682,A -85,B 0,C 180,E1 -15365.299,E2 -15365.299} C_VEL
LIN {X 0,Y 319.563,Z 310.678,A -85,B 0,C 180,E1 -15368.046,E2 -15368.046} C_VEL
LIN {X 0,Y 319.623,Z 310.671,A -85,B 0,C 180,E1 -15372.072,E2 -15372.072} C_VEL
LIN {X 0,Y 319.736,Z 310.822,A -85,B 0,C 180,E1 -15374.755,E2 -15374.755} C_VEL
LIN {X 0,Y 320.826,Z 316.047,A -85,B 0,C 180,E1 -15376.315,E2 -15376.315} C_VEL
LIN {X 0,Y 326.556,Z 333.056,A -85,B 0,C 180,E1 -15377.098,E2 -15377.098} C_VEL
LIN {X 0,Y 328.558,Z 344.833,A -85,B 0,C 180,E1 -15377.492,E2 -15377.492} C_VEL
LIN {X 0,Y 326.904,Z 424.072,A -85,B 0,C 180,E1 -15379.236,E2 -15379.236} C_VEL
LIN {X 0,Y 326.32,Z 437.776,A -85,B 0,C 180,E1 -15379.805,E2 -15379.805} C_VEL
LIN {X 0,Y 325.586,Z 450.594,A -85,B 0,C 180,E1 -15380.605,E2 -15380.605} C_VEL
LIN {X 0,Y 324.687,Z 462.284,A -85,B 0,C 180,E1 -15381.599,E2 -15381.599} C_VEL
LIN {X 0,Y 323.29,Z 473.627,A -85,B 0,C 180,E1 -15382.82,E2 -15382.82} C_VEL
LIN {X 0,Y 322.242,Z 483.786,A -85,B 0,C 180,E1 -15384.211,E2 -15384.211} C_VEL
LIN {X 0,Y 321.061,Z 493.741,A -85,B 0,C 180,E1 -15385.921,E2 -15385.921} C_VEL
LIN {X 0,Y 320.088,Z 502.497,A -85,B 0,C 180,E1 -15387.798,E2 -15387.798} C_VEL
LIN {X 0,Y 319.179,Z 509.531,A -85,B 0,C 180,E1 -15389.685,E2 -15389.685} C_VEL
LIN {X 0,Y 318.6,Z 515.936,A -85,B 0,C 180,E1 -15391.897,E2 -15391.897} C_VEL
LIN {X 0,Y 318.179,Z 520.179,A -85,B 0,C 180,E1 -15393.8,E2 -15393.8} C_VEL
LIN {X 0,Y 318.074,Z 523.94,A -85,B 0,C 180,E1 -15396.123,E2 -15396.123} C_VEL
LIN {X 0,Y 317.849,Z 525.571,A -85,B 0,C 180,E1 -15397.624,E2 -15397.624} C_VEL
LIN {X 0,Y 317.727,Z 526.535,A -85,B 0,C 180,E1 -15398.908,E2 -15398.908} C_VEL
LIN {X 0,Y 317.675,Z 527.109,A -85,B 0,C 180,E1 -15400.195,E2 -15400.195} C_VEL
LIN {X 0,Y 317.763,Z 527.24,A -85,B 0,C 180,E1 -15401.482,E2 -15401.482} C_VEL
LIN {X 0,Y 318.007,Z 526.663,A -85,B 0,C 180,E1 -15403.492,E2 -15403.492} C_VEL
LIN {X 0,Y 318.233,Z 525.246,A -85,B 0,C 180,E1 -15405.368,E2 -15405.368} C_VEL
LIN {X 0,Y 318.517,Z 523.711,A -85,B 0,C 180,E1 -15406.669,E2 -15406.669} C_VEL
LIN {X 0,Y 319.208,Z 520.273,A -85,B 0,C 180,E1 -15408.786,E2 -15408.786} C_VEL
LIN {X 0,Y 319.98,Z 516.36,A -85,B 0,C 180,E1 -15410.575,E2 -15410.575} C_VEL
LIN {X 0,Y 321.283,Z 509.861,A -85,B 0,C 180,E1 -15412.848,E2 -15412.848} C_VEL
LIN {X 0,Y 322.638,Z 502.676,A -85,B 0,C 180,E1 -15414.792,E2 -15414.792} C_VEL
LIN {X 0,Y 324.374,Z 493.632,A -85,B 0,C 180,E1 -15416.717,E2 -15416.717} C_VEL
LIN {X 0,Y 326.056,Z 484.298,A -85,B 0,C 180,E1 -15418.308,E2 -15418.308} C_VEL
LIN {X 0,Y 327.72,Z 473.82,A -85,B 0,C 180,E1 -15419.731,E2 -15419.731} C_VEL
LIN {X 0,Y 329.105,Z 463.723,A -85,B 0,C 180,E1 -15420.832,E2 -15420.832} C_VEL
LIN {X 0,Y 330.536,Z 451.182,A -85,B 0,C 180,E1 -15421.9,E2 -15421.9} C_VEL
LIN {X 0,Y 331.548,Z 438.841,A -85,B 0,C 180,E1 -15422.675,E2 -15422.675} C_VEL
LIN {X 0,Y 332.174,Z 425.853,A -85,B 0,C 180,E1 -15423.238,E2 -15423.238} C_VEL
LIN {X 0,Y 332.957,Z 405.2,A -85,B 0,C 180,E1 -15423.72,E2 -15423.72} C_VEL
LIN {X 0,Y 334.569,Z 347.835,A -85,B 0,C 180,E1 -15424.949,E2 -15424.949} C_VEL
LIN {X 0,Y 333.393,Z 343.714,A -85,B 0,C 180,E1 -15425.16,E2 -15425.16} C_VEL
LIN {X 0,Y 330.634,Z 338.964,A -85,B 0,C 180,E1 -15425.541,E2 -15425.541} C_VEL
LIN {X 0,Y 324.626,Z 332.336,A -85,B 0,C 180,E1 -15426.308,E2 -15426.308} C_VEL
LIN {X 0,Y 318.633,Z 325.741,A -85,B 0,C 180,E1 -15427.108,E2 -15427.108} C_VEL
LIN {X 0,Y 315.882,Z 321.035,A -85,B 0,C 180,E1 -15427.532,E2 -15427.532} C_VEL
LIN {X 0,Y 313.897,Z 316.959,A -85,B 0,C 180,E1 -15427.869,E2 -15427.869} C_VEL
LIN {X 0,Y 312.498,Z 311.558,A -85,B 0,C 180,E1 -15429.83,E2 -15429.83} C_VEL
LIN {X 0,Y 312.489,Z 311.558,A -85,B 0,C 180,E1 -15432.432,E2 -15432.432} C_VEL
LIN {X 0,Y 312.458,Z 311.564,A -85,B 0,C 180,E1 -15436.035,E2 -15436.035} C_VEL
LIN {X 0,Y 312.504,Z 311.556,A -85,B 0,C 180,E1 -15439.875,E2 -15439.875} C_VEL
LIN {X 0,Y 312.535,Z 311.549,A -85,B 0,C 180,E1 -15444.051,E2 -15444.051} C_VEL
LIN {X 0,Y 312.504,Z 311.553,A -85,B 0,C 180,E1 -15447.334,E2 -15447.334} C_VEL
LIN {X 0,Y 312.552,Z 311.545,A -85,B 0,C 180,E1 -15451.276,E2 -15451.276} C_VEL
LIN {X 0,Y 312.585,Z 311.542,A -85,B 0,C 180,E1 -15454.711,E2 -15454.711} C_VEL
LIN {X 0,Y 312.537,Z 311.551,A -85,B 0,C 180,E1 -15458.913,E2 -15458.913} C_VEL
LIN {X 0,Y 312.638,Z 311.537,A -85,B 0,C 180,E1 -15461.657,E2 -15461.657} C_VEL
LIN {X 0,Y 312.694,Z 311.53,A -85,B 0,C 180,E1 -15465.686,E2 -15465.686} C_VEL
LIN {X 0,Y 312.702,Z 311.527,A -85,B 0,C 180,E1 -15469.642,E2 -15469.642} C_VEL
LIN {X 0,Y 312.872,Z 311.508,A -85,B 0,C 180,E1 -15472.255,E2 -15472.255} C_VEL
LIN {X 0,Y 312.717,Z 311.527,A -85,B 0,C 180,E1 -15474.843,E2 -15474.843} C_VEL
LIN {X 0,Y 312.989,Z 311.491,A -85,B 0,C 180,E1 -15478.714,E2 -15478.714} C_VEL
LIN {X 0,Y 312.988,Z 311.493,A -85,B 0,C 180,E1 -15481.287,E2 -15481.287} C_VEL
LIN {X 0,Y 312.717,Z 311.527,A -85,B 0,C 180,E1 -15485.158,E2 -15485.158} C_VEL
LIN {X 0,Y 312.872,Z 311.5,A -85,B 0,C 180,E1 -15487.746,E2 -15487.746} C_VEL
LIN {X 0,Y 312.67,Z 311.526,A -85,B 0,C 180,E1 -15491.672,E2 -15491.672} C_VEL
LIN {X 0,Y 312.701,Z 311.527,A -85,B 0,C 180,E1 -15494.888,E2 -15494.888} C_VEL
LIN {X 0,Y 312.63,Z 311.537,A -85,B 0,C 180,E1 -15499.236,E2 -15499.236} C_VEL
LIN {X 0,Y 312.527,Z 311.556,A -85,B 0,C 180,E1 -15502.781,E2 -15502.781} C_VEL
LIN {X 0,Y 312.583,Z 311.55,A -85,B 0,C 180,E1 -15506.723,E2 -15506.723} C_VEL
LIN {X 0,Y 312.546,Z 311.551,A -85,B 0,C 180,E1 -15509.65,E2 -15509.65} C_VEL
LIN {X 0,Y 312.521,Z 311.555,A -85,B 0,C 180,E1 -15513.689,E2 -15513.689} C_VEL
LIN {X 0,Y 312.527,Z 311.556,A -85,B 0,C 180,E1 -15517.385,E2 -15517.385} C_VEL
LIN {X 0,Y 312.491,Z 311.535,A -85,B 0,C 180,E1 -15520.709,E2 -15520.709} C_VEL
LIN {X 0,Y 312.453,Z 311.56,A -85,B 0,C 180,E1 -15524.21,E2 -15524.21} C_VEL
LIN {X 0,Y 312.486,Z 311.562,A -85,B 0,C 180,E1 -15527.919,E2 -15527.919} C_VEL
LIN {X 0,Y 312.507,Z 311.555,A -85,B 0,C 180,E1 -15531.917,E2 -15531.917} C_VEL
LIN {X 0,Y 312.567,Z 311.726,A -85,B 0,C 180,E1 -15534.621,E2 -15534.621} C_VEL
LIN {X 0,Y 315.551,Z 323.527,A -85,B 0,C 180,E1 -15538.537,E2 -15538.537} C_VEL
LIN {X 0,Y 317.726,Z 333.419,A -85,B 0,C 180,E1 -15541.603,E2 -15541.603} C_VEL
LIN {X 0,Y 318.45,Z 337.241,A -85,B 0,C 180,E1 -15542.704,E2 -15542.704} C_VEL
LIN {X 0,Y 320.21,Z 342.404,A -85,B 0,C 180,E1 -15543.024,E2 -15543.024} C_VEL
LIN {X 0,Y 325.435,Z 367.783,A -85,B 0,C 180,E1 -15544.196,E2 -15544.196} C_VEL
LIN {X 0,Y 327.507,Z 381.17,A -85,B 0,C 180,E1 -15544.728,E2 -15544.728} C_VEL
LIN {X 0,Y 325.728,Z 445.874,A -85,B 0,C 180,E1 -15546.179,E2 -15546.179} C_VEL
LIN {X 0,Y 324.78,Z 459.057,A -85,B 0,C 180,E1 -15546.697,E2 -15546.697} C_VEL
LIN {X 0,Y 323.505,Z 471.172,A -85,B 0,C 180,E1 -15547.402,E2 -15547.402} C_VEL
LIN {X 0,Y 321.989,Z 483.415,A -85,B 0,C 180,E1 -15548.387,E2 -15548.387} C_VEL
LIN {X 0,Y 320.105,Z 494.987,A -85,B 0,C 180,E1 -15549.602,E2 -15549.602} C_VEL
LIN {X 0,Y 318.298,Z 505.41,A -85,B 0,C 180,E1 -15550.993,E2 -15550.993} C_VEL
LIN {X 0,Y 316.436,Z 515.159,A -85,B 0,C 180,E1 -15552.619,E2 -15552.619} C_VEL
LIN {X 0,Y 314.877,Z 523.917,A -85,B 0,C 180,E1 -15554.464,E2 -15554.464} C_VEL
LIN {X 0,Y 313.448,Z 531.266,A -85,B 0,C 180,E1 -15556.383,E2 -15556.383} C_VEL
LIN {X 0,Y 312.277,Z 537.184,A -85,B 0,C 180,E1 -15558.313,E2 -15558.313} C_VEL
LIN {X 0,Y 311.533,Z 541.876,A -85,B 0,C 180,E1 -15560.259,E2 -15560.259} C_VEL
LIN {X 0,Y 311.028,Z 545.475,A -85,B 0,C 180,E1 -15562.208,E2 -15562.208} C_VEL
LIN {X 0,Y 310.739,Z 548.308,A -85,B 0,C 180,E1 -15564.359,E2 -15564.359} C_VEL
LIN {X 0,Y 310.72,Z 549.758,A -85,B 0,C 180,E1 -15566.109,E2 -15566.109} C_VEL
LIN {X 0,Y 310.7,Z 550.384,A -85,B 0,C 180,E1 -15567.407,E2 -15567.407} C_VEL
LIN {X 0,Y 310.693,Z 550.618,A -85,B 0,C 180,E1 -15568.703,E2 -15568.703} C_VEL
LIN {X 0,Y 310.76,Z 550.42,A -85,B 0,C 180,E1 -15570,E2 -15570} C_VEL
LIN {X 0,Y 310.721,Z 549.824,A -85,B 0,C 180,E1 -15571.296,E2 -15571.296} C_VEL
LIN {X 0,Y 310.723,Z 548.836,A -85,B 0,C 180,E1 -15572.592,E2 -15572.592} C_VEL
LIN {X 0,Y 310.759,Z 547.442,A -85,B 0,C 180,E1 -15573.89,E2 -15573.89} C_VEL
LIN {X 0,Y 310.785,Z 544.679,A -85,B 0,C 180,E1 -15575.728,E2 -15575.728} C_VEL
LIN {X 0,Y 311.002,Z 540.488,A -85,B 0,C 180,E1 -15577.792,E2 -15577.792} C_VEL
LIN {X 0,Y 311.472,Z 534.306,A -85,B 0,C 180,E1 -15580.071,E2 -15580.071} C_VEL
LIN {X 0,Y 312.118,Z 527.541,A -85,B 0,C 180,E1 -15582.021,E2 -15582.021} C_VEL
LIN {X 0,Y 313.139,Z 519.146,A -85,B 0,C 180,E1 -15583.961,E2 -15583.961} C_VEL
LIN {X 0,Y 314.224,Z 510.492,A -85,B 0,C 180,E1 -15585.568,E2 -15585.568} C_VEL
LIN {X 0,Y 315.283,Z 499.775,A -85,B 0,C 180,E1 -15587.178,E2 -15587.178} C_VEL
LIN {X 0,Y 316.493,Z 489.16,A -85,B 0,C 180,E1 -15588.447,E2 -15588.447} C_VEL
LIN {X 0,Y 317.769,Z 477.389,A -85,B 0,C 180,E1 -15589.542,E2 -15589.542} C_VEL
LIN {X 0,Y 318.771,Z 465.111,A -85,B 0,C 180,E1 -15590.402,E2 -15590.402} C_VEL
LIN {X 0,Y 319.674,Z 451.698,A -85,B 0,C 180,E1 -15591.057,E2 -15591.057} C_VEL
LIN {X 0,Y 320.08,Z 438.207,A -85,B 0,C 180,E1 -15591.451,E2 -15591.451} C_VEL
LIN {X 0,Y 321.209,Z 378.632,A -85,B 0,C 180,E1 -15592.768,E2 -15592.768} C_VEL
LIN {X 0,Y 315.634,Z 337.801,A -85,B 0,C 180,E1 -15594.087,E2 -15594.087} C_VEL
LIN {X 0,Y 316.364,Z 331.575,A -85,B 0,C 180,E1 -15595.669,E2 -15595.669} C_VEL
LIN {X 0,Y 315.424,Z 325.301,A -85,B 0,C 180,E1 -15597.388,E2 -15597.388} C_VEL
LIN {X 0,Y 312.968,Z 313.65,A -85,B 0,C 180,E1 -15600.721,E2 -15600.721} C_VEL
LIN {X 0,Y 312.496,Z 311.562,A -85,B 0,C 180,E1 -15601.353,E2 -15601.353} C_VEL
LIN {X 0,Y 312.506,Z 311.561,A -85,B 0,C 180,E1 -15604.209,E2 -15604.209} C_VEL
LIN {X 0,Y 312.533,Z 311.555,A -85,B 0,C 180,E1 -15608.089,E2 -15608.089} C_VEL
LIN {X 0,Y 312.483,Z 311.561,A -85,B 0,C 180,E1 -15612.081,E2 -15612.081} C_VEL
LIN {X 0,Y 312.456,Z 311.563,A -85,B 0,C 180,E1 -15616.034,E2 -15616.034} C_VEL
LIN {X 0,Y 312.502,Z 311.556,A -85,B 0,C 180,E1 -15619.874,E2 -15619.874} C_VEL
LIN {X 0,Y 312.533,Z 311.553,A -85,B 0,C 180,E1 -15624.05,E2 -15624.05} C_VEL
LIN {X 0,Y 312.501,Z 311.557,A -85,B 0,C 180,E1 -15627.333,E2 -15627.333} C_VEL
LIN {X 0,Y 312.541,Z 311.553,A -85,B 0,C 180,E1 -15631.278,E2 -15631.278} C_VEL
LIN {X 0,Y 312.582,Z 311.548,A -85,B 0,C 180,E1 -15634.71,E2 -15634.71} C_VEL
LIN {X 0,Y 312.584,Z 311.547,A -85,B 0,C 180,E1 -15637.528,E2 -15637.528} C_VEL
LIN {X 0,Y 312.635,Z 311.54,A -85,B 0,C 180,E1 -15641.656,E2 -15641.656} C_VEL
LIN {X 0,Y 312.69,Z 311.533,A -85,B 0,C 180,E1 -15645.686,E2 -15645.686} C_VEL
LIN {X 0,Y 312.697,Z 311.532,A -85,B 0,C 180,E1 -15649.641,E2 -15649.641} C_VEL
LIN {X 0,Y 312.862,Z 311.51,A -85,B 0,C 180,E1 -15652.254,E2 -15652.254} C_VEL
LIN {X 0,Y 312.711,Z 311.529,A -85,B 0,C 180,E1 -15654.842,E2 -15654.842} C_VEL
LIN {X 0,Y 312.986,Z 311.49,A -85,B 0,C 180,E1 -15658.713,E2 -15658.713} C_VEL
LIN {X 0,Y 312.984,Z 311.494,A -85,B 0,C 180,E1 -15661.286,E2 -15661.286} C_VEL
LIN {X 0,Y 312.703,Z 311.531,A -85,B 0,C 180,E1 -15665.158,E2 -15665.158} C_VEL
LIN {X 0,Y 312.813,Z 311.519,A -85,B 0,C 180,E1 -15667.747,E2 -15667.747} C_VEL
LIN {X 0,Y 312.664,Z 311.534,A -85,B 0,C 180,E1 -15671.671,E2 -15671.671} C_VEL
LIN {X 0,Y 312.695,Z 311.531,A -85,B 0,C 180,E1 -15674.888,E2 -15674.888} C_VEL
LIN {X 0,Y 312.604,Z 311.539,A -85,B 0,C 180,E1 -15679.225,E2 -15679.225} C_VEL
LIN {X 0,Y 312.521,Z 311.554,A -85,B 0,C 180,E1 -15682.78,E2 -15682.78} C_VEL
LIN {X 0,Y 312.598,Z 311.545,A -85,B 0,C 180,E1 -15685.936,E2 -15685.936} C_VEL
LIN {X 0,Y 312.54,Z 311.546,A -85,B 0,C 180,E1 -15689.65,E2 -15689.65} C_VEL
LIN {X 0,Y 312.515,Z 311.553,A -85,B 0,C 180,E1 -15693.689,E2 -15693.689} C_VEL
LIN {X 0,Y 312.515,Z 311.551,A -85,B 0,C 180,E1 -15697.386,E2 -15697.386} C_VEL
LIN {X 0,Y 312.486,Z 311.559,A -85,B 0,C 180,E1 -15700.71,E2 -15700.71} C_VEL
LIN {X 0,Y 312.447,Z 311.561,A -85,B 0,C 180,E1 -15704.21,E2 -15704.21} C_VEL
LIN {X 0,Y 312.451,Z 311.561,A -85,B 0,C 180,E1 -15707.925,E2 -15707.925} C_VEL
LIN {X 0,Y 312.48,Z 311.556,A -85,B 0,C 180,E1 -15711.923,E2 -15711.923} C_VEL
LIN {X 0,Y 312.527,Z 311.552,A -85,B 0,C 180,E1 -15714.221,E2 -15714.221} C_VEL
LIN {X 0,Y 312.498,Z 311.561,A -85,B 0,C 180,E1 -15717.334,E2 -15717.334} C_VEL
LIN {X 0,Y 312.495,Z 311.559,A -85,B 0,C 180,E1 -15721.295,E2 -15721.295} C_VEL
LIN {X 0,Y 312.519,Z 311.553,A -85,B 0,C 180,E1 -15724.706,E2 -15724.706} C_VEL
LIN {X 0,Y 312.559,Z 311.554,A -85,B 0,C 180,E1 -15727.528,E2 -15727.528} C_VEL
LIN {X 0,Y 312.58,Z 311.551,A -85,B 0,C 180,E1 -15731.654,E2 -15731.654} C_VEL
LIN {X 0,Y 312.669,Z 311.638,A -85,B 0,C 180,E1 -15734.403,E2 -15734.403} C_VEL
LIN {X 0,Y 313.63,Z 316.311,A -85,B 0,C 180,E1 -15735.833,E2 -15735.833} C_VEL
LIN {X 0,Y 319.646,Z 333.773,A -85,B 0,C 180,E1 -15736.672,E2 -15736.672} C_VEL
LIN {X 0,Y 321.847,Z 345.396,A -85,B 0,C 180,E1 -15737.087,E2 -15737.087} C_VEL
LIN {X 0,Y 320.162,Z 423.974,A -85,B 0,C 180,E1 -15738.847,E2 -15738.847} C_VEL
LIN {X 0,Y 319.602,Z 437.043,A -85,B 0,C 180,E1 -15739.388,E2 -15739.388} C_VEL
LIN {X 0,Y 318.884,Z 449.623,A -85,B 0,C 180,E1 -15740.166,E2 -15740.166} C_VEL
LIN {X 0,Y 318,Z 460.854,A -85,B 0,C 180,E1 -15741.101,E2 -15741.101} C_VEL
LIN {X 0,Y 317.062,Z 468.457,A -85,B 0,C 180,E1 -15741.877,E2 -15741.877} C_VEL
LIN {X 0,Y 315.925,Z 478.577,A -85,B 0,C 180,E1 -15743.133,E2 -15743.133} C_VEL
LIN {X 0,Y 314.851,Z 487.871,A -85,B 0,C 180,E1 -15744.557,E2 -15744.557} C_VEL
LIN {X 0,Y 313.86,Z 496.344,A -85,B 0,C 180,E1 -15746.149,E2 -15746.149} C_VEL
LIN {X 0,Y 312.831,Z 504.6,A -85,B 0,C 180,E1 -15748.069,E2 -15748.069} C_VEL
LIN {X 0,Y 311.989,Z 511.263,A -85,B 0,C 180,E1 -15750,E2 -15750} C_VEL
LIN {X 0,Y 311.503,Z 516.574,A -85,B 0,C 180,E1 -15751.94,E2 -15751.94} C_VEL
LIN {X 0,Y 311.098,Z 520.73,A -85,B 0,C 180,E1 -15753.886,E2 -15753.886} C_VEL
LIN {X 0,Y 311.005,Z 524.217,A -85,B 0,C 180,E1 -15756.123,E2 -15756.123} C_VEL
LIN {X 0,Y 310.739,Z 525.968,A -85,B 0,C 180,E1 -15757.8,E2 -15757.8} C_VEL
LIN {X 0,Y 310.628,Z 526.896,A -85,B 0,C 180,E1 -15759.113,E2 -15759.113} C_VEL
